LIN {X 0,Y 372.523,Z 405.276,A -85,B 0,C 180,E1 -12705.139,E2 -12705.139} C_VEL
LIN {X 0,Y 373,Z 395.69,A -85,B 0,C 180,E1 -12705.477,E2 -12705.477} C_VEL
LIN {X 0,Y 373.56,Z 352.776,A -85,B 0,C 180,E1 -12706.364,E2 -12706.364} C_VEL
LIN {X 0,Y 373.405,Z 343.149,A -85,B 0,C 180,E1 -12706.57,E2 -12706.57} C_VEL
LIN {X 0,Y 370.133,Z 321.024,A -85,B 0,C 180,E1 -12707.194,E2 -12707.194} C_VEL
LIN {X 0,Y 369.546,Z 317.373,A -85,B 0,C 180,E1 -12707.322,E2 -12707.322} C_VEL
LIN {X 0,Y 370.614,Z 302.559,A -85,B 0,C 180,E1 -12711.118,E2 -12711.118} C_VEL
LIN {X 0,Y 371.037,Z 295.89,A -85,B 0,C 180,E1 -12712.848,E2 -12712.848} C_VEL
LIN {X 0,Y 369.464,Z 286.97,A -85,B 0,C 180,E1 -12715.34,E2 -12715.34} C_VEL
LIN {X 0,Y 368.919,Z 284.344,A -85,B 0,C 180,E1 -12716.097,E2 -12716.097} C_VEL
LIN {X 0,Y 368.891,Z 284.349,A -85,B 0,C 180,E1 -12719.691,E2 -12719.691} C_VEL
LIN {X 0,Y 368.893,Z 284.348,A -85,B 0,C 180,E1 -12723.042,E2 -12723.042} C_VEL
LIN {X 0,Y 368.912,Z 284.344,A -85,B 0,C 180,E1 -12726.196,E2 -12726.196} C_VEL
LIN {X 0,Y 368.896,Z 284.351,A -85,B 0,C 180,E1 -12728.953,E2 -12728.953} C_VEL
LIN {X 0,Y 368.874,Z 284.348,A -85,B 0,C 180,E1 -12732.008,E2 -12732.008} C_VEL
LIN {X 0,Y 368.873,Z 284.351,A -85,B 0,C 180,E1 -12735.175,E2 -12735.175} C_VEL
LIN {X 0,Y 368.875,Z 284.345,A -85,B 0,C 180,E1 -12738.177,E2 -12738.177} C_VEL
LIN {X 0,Y 368.899,Z 284.348,A -85,B 0,C 180,E1 -12741.359,E2 -12741.359} C_VEL
LIN {X 0,Y 368.928,Z 284.341,A -85,B 0,C 180,E1 -12745.146,E2 -12745.146} C_VEL
LIN {X 0,Y 368.921,Z 284.338,A -85,B 0,C 180,E1 -12749.046,E2 -12749.046} C_VEL
LIN {X 0,Y 368.966,Z 284.335,A -85,B 0,C 180,E1 -12751.563,E2 -12751.563} C_VEL
LIN {X 0,Y 368.99,Z 284.33,A -85,B 0,C 180,E1 -12754.019,E2 -12754.019} C_VEL
LIN {X 0,Y 368.911,Z 284.338,A -85,B 0,C 180,E1 -12757.604,E2 -12757.604} C_VEL
LIN {X 0,Y 368.947,Z 284.337,A -85,B 0,C 180,E1 -12761.105,E2 -12761.105} C_VEL
LIN {X 0,Y 368.986,Z 284.325,A -85,B 0,C 180,E1 -12764.535,E2 -12764.535} C_VEL
LIN {X 0,Y 368.994,Z 284.332,A -85,B 0,C 180,E1 -12767.906,E2 -12767.906} C_VEL
LIN {X 0,Y 369.156,Z 284.304,A -85,B 0,C 180,E1 -12771.869,E2 -12771.869} C_VEL
LIN {X 0,Y 369.13,Z 284.317,A -85,B 0,C 180,E1 -12774.537,E2 -12774.537} C_VEL
LIN {X 0,Y 369.304,Z 284.286,A -85,B 0,C 180,E1 -12777.819,E2 -12777.819} C_VEL
LIN {X 0,Y 369.446,Z 284.273,A -85,B 0,C 180,E1 -12780,E2 -12780} C_VEL
LIN {X 0,Y 369.305,Z 284.283,A -85,B 0,C 180,E1 -12782.181,E2 -12782.181} C_VEL
LIN {X 0,Y 369.161,Z 284.309,A -85,B 0,C 180,E1 -12786.559,E2 -12786.559} C_VEL
LIN {X 0,Y 369.056,Z 284.325,A -85,B 0,C 180,E1 -12789.869,E2 -12789.869} C_VEL
LIN {X 0,Y 369.027,Z 284.331,A -85,B 0,C 180,E1 -12793.773,E2 -12793.773} C_VEL
LIN {X 0,Y 368.992,Z 284.336,A -85,B 0,C 180,E1 -12797.769,E2 -12797.769} C_VEL
LIN {X 0,Y 368.92,Z 284.341,A -85,B 0,C 180,E1 -12801.22,E2 -12801.22} C_VEL
LIN {X 0,Y 368.949,Z 284.339,A -85,B 0,C 180,E1 -12804.776,E2 -12804.776} C_VEL
LIN {X 0,Y 368.978,Z 284.334,A -85,B 0,C 180,E1 -12808.436,E2 -12808.436} C_VEL
LIN {X 0,Y 368.891,Z 284.349,A -85,B 0,C 180,E1 -12812.239,E2 -12812.239} C_VEL
LIN {X 0,Y 368.922,Z 284.338,A -85,B 0,C 180,E1 -12815.002,E2 -12815.002} C_VEL
LIN {X 0,Y 368.906,Z 284.346,A -85,B 0,C 180,E1 -12818.642,E2 -12818.642} C_VEL
LIN {X 0,Y 368.956,Z 284.341,A -85,B 0,C 180,E1 -12820.813,E2 -12820.813} C_VEL
LIN {X 0,Y 370.249,Z 291.31,A -85,B 0,C 180,E1 -12822.819,E2 -12822.819} C_VEL
LIN {X 0,Y 369.978,Z 298.523,A -85,B 0,C 180,E1 -12824.755,E2 -12824.755} C_VEL
LIN {X 0,Y 373.924,Z 318.904,A -85,B 0,C 180,E1 -12825.4,E2 -12825.4} C_VEL
LIN {X 0,Y 373.092,Z 375.949,A -85,B 0,C 180,E1 -12826.565,E2 -12826.565} C_VEL
LIN {X 0,Y 372.739,Z 386.647,A -85,B 0,C 180,E1 -12826.954,E2 -12826.954} C_VEL
LIN {X 0,Y 372.199,Z 398.56,A -85,B 0,C 180,E1 -12827.636,E2 -12827.636} C_VEL
LIN {X 0,Y 371.586,Z 407.896,A -85,B 0,C 180,E1 -12828.37,E2 -12828.37} C_VEL
LIN {X 0,Y 370.993,Z 415.935,A -85,B 0,C 180,E1 -12829.168,E2 -12829.168} C_VEL
LIN {X 0,Y 370.411,Z 422.879,A -85,B 0,C 180,E1 -12830.006,E2 -12830.006} C_VEL
LIN {X 0,Y 369.807,Z 429.621,A -85,B 0,C 180,E1 -12830.986,E2 -12830.986} C_VEL
LIN {X 0,Y 369.35,Z 434.404,A -85,B 0,C 180,E1 -12831.801,E2 -12831.801} C_VEL
LIN {X 0,Y 368.78,Z 440.973,A -85,B 0,C 180,E1 -12833.17,E2 -12833.17} C_VEL
LIN {X 0,Y 368.379,Z 445.802,A -85,B 0,C 180,E1 -12834.418,E2 -12834.418} C_VEL
LIN {X 0,Y 367.918,Z 449.947,A -85,B 0,C 180,E1 -12835.759,E2 -12835.759} C_VEL
LIN {X 0,Y 367.739,Z 453.397,A -85,B 0,C 180,E1 -12837.236,E2 -12837.236} C_VEL
LIN {X 0,Y 367.446,Z 456.117,A -85,B 0,C 180,E1 -12838.909,E2 -12838.909} C_VEL
LIN {X 0,Y 367.291,Z 457.289,A -85,B 0,C 180,E1 -12840.166,E2 -12840.166} C_VEL
LIN {X 0,Y 367.214,Z 457.874,A -85,B 0,C 180,E1 -12841.689,E2 -12841.689} C_VEL
LIN {X 0,Y 367.2,Z 457.67,A -85,B 0,C 180,E1 -12842.656,E2 -12842.656} C_VEL
LIN {X 0,Y 367.282,Z 456.753,A -85,B 0,C 180,E1 -12844.074,E2 -12844.074} C_VEL
LIN {X 0,Y 367.469,Z 454.638,A -85,B 0,C 180,E1 -12845.721,E2 -12845.721} C_VEL
LIN {X 0,Y 367.777,Z 450.863,A -85,B 0,C 180,E1 -12847.532,E2 -12847.532} C_VEL
LIN {X 0,Y 368.018,Z 447.468,A -85,B 0,C 180,E1 -12848.726,E2 -12848.726} C_VEL
LIN {X 0,Y 368.416,Z 442.007,A -85,B 0,C 180,E1 -12850.209,E2 -12850.209} C_VEL
LIN {X 0,Y 368.818,Z 436.622,A -85,B 0,C 180,E1 -12851.388,E2 -12851.388} C_VEL
LIN {X 0,Y 369.347,Z 430.05,A -85,B 0,C 180,E1 -12852.561,E2 -12852.561} C_VEL
LIN {X 0,Y 369.885,Z 423.088,A -85,B 0,C 180,E1 -12853.583,E2 -12853.583} C_VEL
LIN {X 0,Y 370.406,Z 415.905,A -85,B 0,C 180,E1 -12854.455,E2 -12854.455} C_VEL
LIN {X 0,Y 370.966,Z 408.076,A -85,B 0,C 180,E1 -12855.234,E2 -12855.234} C_VEL
LIN {X 0,Y 371.424,Z 399.77,A -85,B 0,C 180,E1 -12855.9,E2 -12855.9} C_VEL
LIN {X 0,Y 371.823,Z 390.588,A -85,B 0,C 180,E1 -12856.473,E2 -12856.473} C_VEL
LIN {X 0,Y 372.259,Z 379.24,A -85,B 0,C 180,E1 -12856.976,E2 -12856.976} C_VEL
LIN {X 0,Y 372.545,Z 362.521,A -85,B 0,C 180,E1 -12857.367,E2 -12857.367} C_VEL
LIN {X 0,Y 372.968,Z 318.576,A -85,B 0,C 180,E1 -12858.237,E2 -12858.237} C_VEL
LIN {X 0,Y 369.543,Z 298.791,A -85,B 0,C 180,E1 -12858.8,E2 -12858.8} C_VEL
LIN {X 0,Y 369.932,Z 290.475,A -85,B 0,C 180,E1 -12861.258,E2 -12861.258} C_VEL
LIN {X 0,Y 369.217,Z 284.308,A -85,B 0,C 180,E1 -12863.168,E2 -12863.168} C_VEL
LIN {X 0,Y 369.318,Z 284.296,A -85,B 0,C 180,E1 -12867.819,E2 -12867.819} C_VEL
LIN {X 0,Y 369.459,Z 284.278,A -85,B 0,C 180,E1 -12870,E2 -12870} C_VEL
LIN {X 0,Y 369.319,Z 284.294,A -85,B 0,C 180,E1 -12872.181,E2 -12872.181} C_VEL
LIN {X 0,Y 369.18,Z 284.309,A -85,B 0,C 180,E1 -12876.558,E2 -12876.558} C_VEL
LIN {X 0,Y 369.068,Z 284.323,A -85,B 0,C 180,E1 -12879.868,E2 -12879.868} C_VEL
LIN {X 0,Y 369.038,Z 284.325,A -85,B 0,C 180,E1 -12883.772,E2 -12883.772} C_VEL
LIN {X 0,Y 369.01,Z 284.333,A -85,B 0,C 180,E1 -12884.425,E2 -12884.425} C_VEL
LIN {X 0,Y 368.294,Z 284.417,A -85,B 0,C 180,E1 -12885.335,E2 -12885.335} C_VEL
LIN {X 0,Y 365.388,Z 284.782,A -85,B 0,C 180,E1 -12886.815,E2 -12886.815} C_VEL
LIN {X 0,Y 362.968,Z 285.082,A -85,B 0,C 180,E1 -12888.013,E2 -12888.013} C_VEL
LIN {X 0,Y 361.955,Z 285.21,A -85,B 0,C 180,E1 -12888.939,E2 -12888.939} C_VEL
LIN {X 0,Y 361.885,Z 285.216,A -85,B 0,C 180,E1 -12889.253,E2 -12889.253} C_VEL
LIN {X 0,Y 361.882,Z 285.221,A -85,B 0,C 180,E1 -12892.855,E2 -12892.855} C_VEL
LIN {X 0,Y 361.94,Z 285.214,A -85,B 0,C 180,E1 -12896.721,E2 -12896.721} C_VEL
LIN {X 0,Y 361.873,Z 285.218,A -85,B 0,C 180,E1 -12900.327,E2 -12900.327} C_VEL
LIN {X 0,Y 361.851,Z 285.22,A -85,B 0,C 180,E1 -12904.28,E2 -12904.28} C_VEL
LIN {X 0,Y 361.86,Z 285.226,A -85,B 0,C 180,E1 -12907.222,E2 -12907.222} C_VEL
LIN {X 0,Y 361.832,Z 285.223,A -85,B 0,C 180,E1 -12910.754,E2 -12910.754} C_VEL
LIN {X 0,Y 361.841,Z 285.221,A -85,B 0,C 180,E1 -12914.363,E2 -12914.363} C_VEL
LIN {X 0,Y 361.884,Z 285.222,A -85,B 0,C 180,E1 -12917.558,E2 -12917.558} C_VEL
LIN {X 0,Y 361.868,Z 285.218,A -85,B 0,C 180,E1 -12920.972,E2 -12920.972} C_VEL
LIN {X 0,Y 361.868,Z 285.218,A -85,B 0,C 180,E1 -12924.654,E2 -12924.654} C_VEL
LIN {X 0,Y 361.831,Z 285.225,A -85,B 0,C 180,E1 -12928.37,E2 -12928.37} C_VEL
LIN {X 0,Y 361.894,Z 285.214,A -85,B 0,C 180,E1 -12930.955,E2 -12930.955} C_VEL
LIN {X 0,Y 361.946,Z 285.208,A -85,B 0,C 180,E1 -12933.474,E2 -12933.474} C_VEL
LIN {X 0,Y 361.881,Z 285.216,A -85,B 0,C 180,E1 -12937.144,E2 -12937.144} C_VEL
LIN {X 0,Y 361.895,Z 285.218,A -85,B 0,C 180,E1 -12940.723,E2 -12940.723} C_VEL
LIN {X 0,Y 361.923,Z 285.212,A -85,B 0,C 180,E1 -12943.065,E2 -12943.065} C_VEL
LIN {X 0,Y 361.989,Z 285.208,A -85,B 0,C 180,E1 -12946.527,E2 -12946.527} C_VEL
LIN {X 0,Y 362.021,Z 285.199,A -85,B 0,C 180,E1 -12949.938,E2 -12949.938} C_VEL
LIN {X 0,Y 362.151,Z 285.184,A -85,B 0,C 180,E1 -12953.313,E2 -12953.313} C_VEL
LIN {X 0,Y 362.271,Z 285.168,A -85,B 0,C 180,E1 -12957.776,E2 -12957.776} C_VEL
LIN {X 0,Y 362.416,Z 285.149,A -85,B 0,C 180,E1 -12960,E2 -12960} C_VEL
LIN {X 0,Y 362.269,Z 285.167,A -85,B 0,C 180,E1 -12962.223,E2 -12962.223} C_VEL
LIN {X 0,Y 362.151,Z 285.183,A -85,B 0,C 180,E1 -12966.686,E2 -12966.686} C_VEL
LIN {X 0,Y 362.024,Z 285.199,A -85,B 0,C 180,E1 -12970.062,E2 -12970.062} C_VEL
LIN {X 0,Y 361.988,Z 285.206,A -85,B 0,C 180,E1 -12973.899,E2 -12973.899} C_VEL
LIN {X 0,Y 361.958,Z 285.211,A -85,B 0,C 180,E1 -12977.939,E2 -12977.939} C_VEL
LIN {X 0,Y 361.871,Z 285.221,A -85,B 0,C 180,E1 -12981.654,E2 -12981.654} C_VEL
LIN {X 0,Y 361.917,Z 285.212,A -85,B 0,C 180,E1 -12985.291,E2 -12985.291} C_VEL
LIN {X 0,Y 361.899,Z 285.217,A -85,B 0,C 180,E1 -12987.78,E2 -12987.78} C_VEL
LIN {X 0,Y 361.829,Z 285.223,A -85,B 0,C 180,E1 -12991.63,E2 -12991.63} C_VEL
LIN {X 0,Y 361.866,Z 285.218,A -85,B 0,C 180,E1 -12995.345,E2 -12995.345} C_VEL
LIN {X 0,Y 361.86,Z 285.22,A -85,B 0,C 180,E1 -12999.027,E2 -12999.027} C_VEL
LIN {X 0,Y 361.829,Z 285.227,A -85,B 0,C 180,E1 -13002.83,E2 -13002.83} C_VEL
LIN {X 0,Y 361.813,Z 285.225,A -85,B 0,C 180,E1 -13005.947,E2 -13005.947} C_VEL
LIN {X 0,Y 361.829,Z 285.225,A -85,B 0,C 180,E1 -13009.246,E2 -13009.246} C_VEL
LIN {X 0,Y 361.858,Z 285.223,A -85,B 0,C 180,E1 -13012.778,E2 -13012.778} C_VEL
LIN {X 0,Y 361.85,Z 285.221,A -85,B 0,C 180,E1 -13015.72,E2 -13015.72} C_VEL
LIN {X 0,Y 361.861,Z 285.22,A -85,B 0,C 180,E1 -13019.672,E2 -13019.672} C_VEL
LIN {X 0,Y 361.874,Z 285.222,A -85,B 0,C 180,E1 -13023.78,E2 -13023.78} C_VEL
LIN {X 0,Y 361.907,Z 285.404,A -85,B 0,C 180,E1 -13023.938,E2 -13023.938} C_VEL
LIN {X 0,Y 363.844,Z 295.855,A -85,B 0,C 180,E1 -13026.975,E2 -13026.975} C_VEL
LIN {X 0,Y 363.495,Z 302.362,A -85,B 0,C 180,E1 -13028.746,E2 -13028.746} C_VEL
LIN {X 0,Y 362.389,Z 316.398,A -85,B 0,C 180,E1 -13032.507,E2 -13032.507} C_VEL
LIN {X 0,Y 362.291,Z 317.88,A -85,B 0,C 180,E1 -13032.902,E2 -13032.902} C_VEL
LIN {X 0,Y 366.001,Z 345.967,A -85,B 0,C 180,E1 -13033.672,E2 -13033.672} C_VEL
LIN {X 0,Y 365.308,Z 395.497,A -85,B 0,C 180,E1 -13034.697,E2 -13034.697} C_VEL
LIN {X 0,Y 364.866,Z 405.848,A -85,B 0,C 180,E1 -13035.071,E2 -13035.071} C_VEL
LIN {X 0,Y 364.198,Z 417.985,A -85,B 0,C 180,E1 -13035.757,E2 -13035.757} C_VEL
LIN {X 0,Y 363.671,Z 426.806,A -85,B 0,C 180,E1 -13036.449,E2 -13036.449} C_VEL
LIN {X 0,Y 363.046,Z 435.21,A -85,B 0,C 180,E1 -13037.279,E2 -13037.279} C_VEL
LIN {X 0,Y 362.479,Z 443.159,A -85,B 0,C 180,E1 -13038.254,E2 -13038.254} C_VEL
LIN {X 0,Y 361.867,Z 450.582,A -85,B 0,C 180,E1 -13039.368,E2 -13039.368} C_VEL
LIN {X 0,Y 361.242,Z 458.107,A -85,B 0,C 180,E1 -13040.764,E2 -13040.764} C_VEL
LIN {X 0,Y 360.844,Z 464.009,A -85,B 0,C 180,E1 -13042.164,E2 -13042.164} C_VEL
LIN {X 0,Y 360.609,Z 467.845,A -85,B 0,C 180,E1 -13043.285,E2 -13043.285} C_VEL
LIN {X 0,Y 360.429,Z 472.249,A -85,B 0,C 180,E1 -13044.966,E2 -13044.966} C_VEL
LIN {X 0,Y 360.318,Z 475.324,A -85,B 0,C 180,E1 -13046.646,E2 -13046.646} C_VEL
LIN {X 0,Y 360.269,Z 476.725,A -85,B 0,C 180,E1 -13047.764,E2 -13047.764} C_VEL
LIN {X 0,Y 360.302,Z 477.636,A -85,B 0,C 180,E1 -13048.882,E2 -13048.882} C_VEL
LIN {X 0,Y 360.357,Z 477.957,A -85,B 0,C 180,E1 -13050,E2 -13050} C_VEL
LIN {X 0,Y 360.301,Z 477.756,A -85,B 0,C 180,E1 -13051.118,E2 -13051.118} C_VEL
LIN {X 0,Y 360.267,Z 477.089,A -85,B 0,C 180,E1 -13052.236,E2 -13052.236} C_VEL
LIN {X 0,Y 360.317,Z 475.947,A -85,B 0,C 180,E1 -13053.354,E2 -13053.354} C_VEL
LIN {X 0,Y 360.424,Z 474.277,A -85,B 0,C 180,E1 -13054.473,E2 -13054.473} C_VEL
LIN {X 0,Y 360.51,Z 470.594,A -85,B 0,C 180,E1 -13056.162,E2 -13056.162} C_VEL
LIN {X 0,Y 360.801,Z 467.472,A -85,B 0,C 180,E1 -13057.274,E2 -13057.274} C_VEL
LIN {X 0,Y 361.128,Z 462.472,A -85,B 0,C 180,E1 -13058.674,E2 -13058.674} C_VEL
LIN {X 0,Y 361.678,Z 456.185,A -85,B 0,C 180,E1 -13060.072,E2 -13060.072} C_VEL
LIN {X 0,Y 362.293,Z 450.045,A -85,B 0,C 180,E1 -13061.185,E2 -13061.185} C_VEL
LIN {X 0,Y 362.863,Z 443.608,A -85,B 0,C 180,E1 -13062.159,E2 -13062.159} C_VEL
LIN {X 0,Y 363.565,Z 435.824,A -85,B 0,C 180,E1 -13063.128,E2 -13063.128} C_VEL
LIN {X 0,Y 364.254,Z 427.639,A -85,B 0,C 180,E1 -13063.956,E2 -13063.956} C_VEL
LIN {X 0,Y 365.019,Z 417.265,A -85,B 0,C 180,E1 -13064.78,E2 -13064.78} C_VEL
LIN {X 0,Y 365.679,Z 405.709,A -85,B 0,C 180,E1 -13065.43,E2 -13065.43} C_VEL
LIN {X 0,Y 366.207,Z 395.084,A -85,B 0,C 180,E1 -13065.811,E2 -13065.811} C_VEL
LIN {X 0,Y 366.788,Z 344.866,A -85,B 0,C 180,E1 -13066.868,E2 -13066.868} C_VEL
LIN {X 0,Y 363.324,Z 321.428,A -85,B 0,C 180,E1 -13067.552,E2 -13067.552} C_VEL
LIN {X 0,Y 362.599,Z 317.17,A -85,B 0,C 180,E1 -13067.701,E2 -13067.701} C_VEL
LIN {X 0,Y 363.744,Z 302.471,A -85,B 0,C 180,E1 -13071.536,E2 -13071.536} C_VEL
LIN {X 0,Y 364.042,Z 296.917,A -85,B 0,C 180,E1 -13073.012,E2 -13073.012} C_VEL
LIN {X 0,Y 362.423,Z 288.013,A -85,B 0,C 180,E1 -13075.56,E2 -13075.56} C_VEL
LIN {X 0,Y 361.86,Z 285.224,A -85,B 0,C 180,E1 -13076.376,E2 -13076.376} C_VEL
LIN {X 0,Y 361.852,Z 285.228,A -85,B 0,C 180,E1 -13080.329,E2 -13080.329} C_VEL
LIN {X 0,Y 361.85,Z 285.223,A -85,B 0,C 180,E1 -13084.28,E2 -13084.28} C_VEL
LIN {X 0,Y 361.858,Z 285.226,A -85,B 0,C 180,E1 -13087.222,E2 -13087.222} C_VEL
LIN {X 0,Y 361.829,Z 285.232,A -85,B 0,C 180,E1 -13090.754,E2 -13090.754} C_VEL
LIN {X 0,Y 361.81,Z 285.23,A -85,B 0,C 180,E1 -13094.368,E2 -13094.368} C_VEL
LIN {X 0,Y 361.829,Z 285.227,A -85,B 0,C 180,E1 -13097.567,E2 -13097.567} C_VEL
LIN {X 0,Y 361.86,Z 285.222,A -85,B 0,C 180,E1 -13100.973,E2 -13100.973} C_VEL
LIN {X 0,Y 361.866,Z 285.219,A -85,B 0,C 180,E1 -13104.655,E2 -13104.655} C_VEL
LIN {X 0,Y 361.829,Z 285.223,A -85,B 0,C 180,E1 -13108.37,E2 -13108.37} C_VEL
LIN {X 0,Y 361.892,Z 285.214,A -85,B 0,C 180,E1 -13110.955,E2 -13110.955} C_VEL
LIN {X 0,Y 361.944,Z 285.202,A -85,B 0,C 180,E1 -13113.474,E2 -13113.474} C_VEL
LIN {X 0,Y 361.869,Z 285.214,A -85,B 0,C 180,E1 -13117.143,E2 -13117.143} C_VEL
LIN {X 0,Y 361.894,Z 285.217,A -85,B 0,C 180,E1 -13120.723,E2 -13120.723} C_VEL
LIN {X 0,Y 361.922,Z 285.207,A -85,B 0,C 180,E1 -13123.066,E2 -13123.066} C_VEL
LIN {X 0,Y 361.988,Z 285.206,A -85,B 0,C 180,E1 -13126.528,E2 -13126.528} C_VEL
LIN {X 0,Y 362.02,Z 285.195,A -85,B 0,C 180,E1 -13129.938,E2 -13129.938} C_VEL
LIN {X 0,Y 362.152,Z 285.183,A -85,B 0,C 180,E1 -13133.314,E2 -13133.314} C_VEL
LIN {X 0,Y 362.268,Z 285.163,A -85,B 0,C 180,E1 -13137.776,E2 -13137.776} C_VEL
LIN {X 0,Y 362.416,Z 285.149,A -85,B 0,C 180,E1 -13140,E2 -13140} C_VEL
LIN {X 0,Y 362.269,Z 285.159,A -85,B 0,C 180,E1 -13142.224,E2 -13142.224} C_VEL
LIN {X 0,Y 362.123,Z 285.187,A -85,B 0,C 180,E1 -13146.687,E2 -13146.687} C_VEL
LIN {X 0,Y 362.02,Z 285.201,A -85,B 0,C 180,E1 -13150.062,E2 -13150.062} C_VEL
LIN {X 0,Y 361.988,Z 285.207,A -85,B 0,C 180,E1 -13153.899,E2 -13153.899} C_VEL
LIN {X 0,Y 361.958,Z 285.213,A -85,B 0,C 180,E1 -13157.939,E2 -13157.939} C_VEL
LIN {X 0,Y 361.883,Z 285.222,A -85,B 0,C 180,E1 -13161.654,E2 -13161.654} C_VEL
LIN {X 0,Y 361.919,Z 285.216,A -85,B 0,C 180,E1 -13165.291,E2 -13165.291} C_VEL
LIN {X 0,Y 361.914,Z 285.218,A -85,B 0,C 180,E1 -13167.779,E2 -13167.779} C_VEL
LIN {X 0,Y 361.839,Z 285.223,A -85,B 0,C 180,E1 -13171.286,E2 -13171.286} C_VEL
LIN {X 0,Y 361.847,Z 285.223,A -85,B 0,C 180,E1 -13174.281,E2 -13174.281} C_VEL
LIN {X 0,Y 361.859,Z 285.223,A -85,B 0,C 180,E1 -13177.224,E2 -13177.224} C_VEL
LIN {X 0,Y 361.958,Z 285.413,A -85,B 0,C 180,E1 -13180.592,E2 -13180.592} C_VEL
LIN {X 0,Y 363.312,Z 292.544,A -85,B 0,C 180,E1 -13182.688,E2 -13182.688} C_VEL
LIN {X 0,Y 363.067,Z 298.691,A -85,B 0,C 180,E1 -13184.372,E2 -13184.372} C_VEL
LIN {X 0,Y 367.17,Z 319.733,A -85,B 0,C 180,E1 -13185.064,E2 -13185.064} C_VEL
LIN {X 0,Y 366.309,Z 376.155,A -85,B 0,C 180,E1 -13186.241,E2 -13186.241} C_VEL
LIN {X 0,Y 365.954,Z 386.701,A -85,B 0,C 180,E1 -13186.632,E2 -13186.632} C_VEL
LIN {X 0,Y 365.456,Z 397.63,A -85,B 0,C 180,E1 -13187.25,E2 -13187.25} C_VEL
LIN {X 0,Y 364.87,Z 406.864,A -85,B 0,C 180,E1 -13187.969,E2 -13187.969} C_VEL
LIN {X 0,Y 364.187,Z 415.457,A -85,B 0,C 180,E1 -13188.817,E2 -13188.817} C_VEL
LIN {X 0,Y 363.563,Z 422.314,A -85,B 0,C 180,E1 -13189.642,E2 -13189.642} C_VEL
LIN {X 0,Y 362.919,Z 428.888,A -85,B 0,C 180,E1 -13190.59,E2 -13190.59} C_VEL
LIN {X 0,Y 362.355,Z 434.922,A -85,B 0,C 180,E1 -13191.638,E2 -13191.638} C_VEL
LIN {X 0,Y 361.791,Z 441.194,A -85,B 0,C 180,E1 -13192.974,E2 -13192.974} C_VEL
LIN {X 0,Y 361.4,Z 445.075,A -85,B 0,C 180,E1 -13193.968,E2 -13193.968} C_VEL
LIN {X 0,Y 361.027,Z 449.08,A -85,B 0,C 180,E1 -13195.215,E2 -13195.215} C_VEL
LIN {X 0,Y 360.766,Z 451.885,A -85,B 0,C 180,E1 -13196.277,E2 -13196.277} C_VEL
LIN {X 0,Y 360.607,Z 454.538,A -85,B 0,C 180,E1 -13197.592,E2 -13197.592} C_VEL
LIN {X 0,Y 360.282,Z 456.997,A -85,B 0,C 180,E1 -13199.525,E2 -13199.525} C_VEL
LIN {X 0,Y 360.117,Z 458.011,A -85,B 0,C 180,E1 -13201.428,E2 -13201.428} C_VEL
LIN {X 0,Y 360.137,Z 457.601,A -85,B 0,C 180,E1 -13203.332,E2 -13203.332} C_VEL
LIN {X 0,Y 360.222,Z 456.505,A -85,B 0,C 180,E1 -13204.583,E2 -13204.583} C_VEL
LIN {X 0,Y 360.514,Z 453.728,A -85,B 0,C 180,E1 -13206.382,E2 -13206.382} C_VEL
LIN {X 0,Y 360.718,Z 450.886,A -85,B 0,C 180,E1 -13207.672,E2 -13207.672} C_VEL
LIN {X 0,Y 361.028,Z 446.618,A -85,B 0,C 180,E1 -13209.132,E2 -13209.132} C_VEL
LIN {X 0,Y 361.382,Z 441.942,A -85,B 0,C 180,E1 -13210.4,E2 -13210.4} C_VEL
LIN {X 0,Y 361.832,Z 436.493,A -85,B 0,C 180,E1 -13211.602,E2 -13211.602} C_VEL
LIN {X 0,Y 362.37,Z 429.854,A -85,B 0,C 180,E1 -13212.799,E2 -13212.799} C_VEL
LIN {X 0,Y 362.917,Z 422.836,A -85,B 0,C 180,E1 -13213.837,E2 -13213.837} C_VEL
LIN {X 0,Y 363.499,Z 415.501,A -85,B 0,C 180,E1 -13214.731,E2 -13214.731} C_VEL
LIN {X 0,Y 364.145,Z 406.579,A -85,B 0,C 180,E1 -13215.612,E2 -13215.612} C_VEL
LIN {X 0,Y 364.748,Z 394.797,A -85,B 0,C 180,E1 -13216.49,E2 -13216.49} C_VEL
LIN {X 0,Y 365.134,Z 385.095,A -85,B 0,C 180,E1 -13217,E2 -13217} C_VEL
LIN {X 0,Y 365.418,Z 376.079,A -85,B 0,C 180,E1 -13217.328,E2 -13217.328} C_VEL
LIN {X 0,Y 365.997,Z 335.574,A -85,B 0,C 180,E1 -13218.175,E2 -13218.175} C_VEL
LIN {X 0,Y 366.158,Z 319.703,A -85,B 0,C 180,E1 -13218.496,E2 -13218.496} C_VEL
LIN {X 0,Y 362.555,Z 298.937,A -85,B 0,C 180,E1 -13219.106,E2 -13219.106} C_VEL
LIN {X 0,Y 362.939,Z 292.344,A -85,B 0,C 180,E1 -13221.089,E2 -13221.089} C_VEL
LIN {X 0,Y 362.186,Z 285.185,A -85,B 0,C 180,E1 -13223.349,E2 -13223.349} C_VEL
LIN {X 0,Y 362.282,Z 285.172,A -85,B 0,C 180,E1 -13227.777,E2 -13227.777} C_VEL
LIN {X 0,Y 362.428,Z 285.154,A -85,B 0,C 180,E1 -13230,E2 -13230} C_VEL
LIN {X 0,Y 362.283,Z 285.17,A -85,B 0,C 180,E1 -13232.223,E2 -13232.223} C_VEL
LIN {X 0,Y 362.141,Z 285.185,A -85,B 0,C 180,E1 -13236.687,E2 -13236.687} C_VEL
LIN {X 0,Y 362.032,Z 285.202,A -85,B 0,C 180,E1 -13240.062,E2 -13240.062} C_VEL
LIN {X 0,Y 361.999,Z 285.203,A -85,B 0,C 180,E1 -13243.898,E2 -13243.898} C_VEL
LIN {X 0,Y 361.929,Z 285.212,A -85,B 0,C 180,E1 -13246.934,E2 -13246.934} C_VEL
LIN {X 0,Y 361.885,Z 285.216,A -85,B 0,C 180,E1 -13249.253,E2 -13249.253} C_VEL
LIN {X 0,Y 361.239,Z 285.301,A -85,B 0,C 180,E1 -13250.182,E2 -13250.182} C_VEL
LIN {X 0,Y 358.356,Z 285.657,A -85,B 0,C 180,E1 -13251.691,E2 -13251.691} C_VEL
LIN {X 0,Y 355.921,Z 285.963,A -85,B 0,C 180,E1 -13252.912,E2 -13252.912} C_VEL
LIN {X 0,Y 354.909,Z 286.085,A -85,B 0,C 180,E1 -13253.858,E2 -13253.858} C_VEL
LIN {X 0,Y 354.845,Z 286.093,A -85,B 0,C 180,E1 -13254.178,E2 -13254.178} C_VEL
LIN {X 0,Y 354.882,Z 286.092,A -85,B 0,C 180,E1 -13257.095,E2 -13257.095} C_VEL
LIN {X 0,Y 354.852,Z 286.092,A -85,B 0,C 180,E1 -13259.678,E2 -13259.678} C_VEL
LIN {X 0,Y 354.804,Z 286.099,A -85,B 0,C 180,E1 -13263.701,E2 -13263.701} C_VEL
LIN {X 0,Y 354.794,Z 286.099,A -85,B 0,C 180,E1 -13266.459,E2 -13266.459} C_VEL
LIN {X 0,Y 354.821,Z 286.101,A -85,B 0,C 180,E1 -13269.423,E2 -13269.423} C_VEL
LIN {X 0,Y 354.786,Z 286.101,A -85,B 0,C 180,E1 -13272.867,E2 -13272.867} C_VEL
LIN {X 0,Y 354.835,Z 286.095,A -85,B 0,C 180,E1 -13276.114,E2 -13276.114} C_VEL
LIN {X 0,Y 354.852,Z 286.093,A -85,B 0,C 180,E1 -13279.188,E2 -13279.188} C_VEL
LIN {X 0,Y 354.803,Z 286.099,A -85,B 0,C 180,E1 -13282.401,E2 -13282.401} C_VEL
LIN {X 0,Y 354.805,Z 286.097,A -85,B 0,C 180,E1 -13284.94,E2 -13284.94} C_VEL
LIN {X 0,Y 354.786,Z 286.102,A -85,B 0,C 180,E1 -13288.404,E2 -13288.404} C_VEL
LIN {X 0,Y 354.846,Z 286.094,A -85,B 0,C 180,E1 -13291.618,E2 -13291.618} C_VEL
LIN {X 0,Y 354.891,Z 286.094,A -85,B 0,C 180,E1 -13294.172,E2 -13294.172} C_VEL
LIN {X 0,Y 354.826,Z 286.097,A -85,B 0,C 180,E1 -13297.893,E2 -13297.893} C_VEL
LIN {X 0,Y 354.913,Z 286.085,A -85,B 0,C 180,E1 -13301.891,E2 -13301.891} C_VEL
LIN {X 0,Y 354.933,Z 286.082,A -85,B 0,C 180,E1 -13305.981,E2 -13305.981} C_VEL
LIN {X 0,Y 354.967,Z 286.077,A -85,B 0,C 180,E1 -13309.735,E2 -13309.735} C_VEL
LIN {X 0,Y 355.115,Z 286.062,A -85,B 0,C 180,E1 -13313.18,E2 -13313.18} C_VEL
LIN {X 0,Y 355.234,Z 286.044,A -85,B 0,C 180,E1 -13317.732,E2 -13317.732} C_VEL
LIN {X 0,Y 355.386,Z 286.025,A -85,B 0,C 180,E1 -13320,E2 -13320} C_VEL
LIN {X 0,Y 355.232,Z 286.044,A -85,B 0,C 180,E1 -13322.268,E2 -13322.268} C_VEL
LIN {X 0,Y 355.114,Z 286.06,A -85,B 0,C 180,E1 -13326.82,E2 -13326.82} C_VEL
LIN {X 0,Y 354.971,Z 286.077,A -85,B 0,C 180,E1 -13330.264,E2 -13330.264} C_VEL
LIN {X 0,Y 354.933,Z 286.084,A -85,B 0,C 180,E1 -13334.019,E2 -13334.019} C_VEL
LIN {X 0,Y 354.913,Z 286.087,A -85,B 0,C 180,E1 -13338.109,E2 -13338.109} C_VEL
LIN {X 0,Y 354.817,Z 286.1,A -85,B 0,C 180,E1 -13342.107,E2 -13342.107} C_VEL
LIN {X 0,Y 354.889,Z 286.091,A -85,B 0,C 180,E1 -13345.828,E2 -13345.828} C_VEL
LIN {X 0,Y 354.809,Z 286.099,A -85,B 0,C 180,E1 -13349.683,E2 -13349.683} C_VEL
LIN {X 0,Y 354.798,Z 286.099,A -85,B 0,C 180,E1 -13353.703,E2 -13353.703} C_VEL
LIN {X 0,Y 354.79,Z 286.105,A -85,B 0,C 180,E1 -13356.46,E2 -13356.46} C_VEL
LIN {X 0,Y 354.817,Z 286.096,A -85,B 0,C 180,E1 -13359.424,E2 -13359.424} C_VEL
LIN {X 0,Y 354.781,Z 286.104,A -85,B 0,C 180,E1 -13362.868,E2 -13362.868} C_VEL
LIN {X 0,Y 354.762,Z 286.104,A -85,B 0,C 180,E1 -13366.104,E2 -13366.104} C_VEL
LIN {X 0,Y 354.781,Z 286.103,A -85,B 0,C 180,E1 -13369.18,E2 -13369.18} C_VEL
LIN {X 0,Y 354.802,Z 286.099,A -85,B 0,C 180,E1 -13372.404,E2 -13372.404} C_VEL
LIN {X 0,Y 354.808,Z 286.103,A -85,B 0,C 180,E1 -13374.942,E2 -13374.942} C_VEL
LIN {X 0,Y 354.789,Z 286.1,A -85,B 0,C 180,E1 -13378.406,E2 -13378.406} C_VEL
LIN {X 0,Y 354.798,Z 286.103,A -85,B 0,C 180,E1 -13381.615,E2 -13381.615} C_VEL
LIN {X 0,Y 354.852,Z 286.176,A -85,B 0,C 180,E1 -13383.696,E2 -13383.696} C_VEL
LIN {X 0,Y 356.803,Z 296.623,A -85,B 0,C 180,E1 -13386.801,E2 -13386.801} C_VEL
LIN {X 0,Y 356.623,Z 302.05,A -85,B 0,C 180,E1 -13388.315,E2 -13388.315} C_VEL
LIN {X 0,Y 355.423,Z 316.087,A -85,B 0,C 180,E1 -13392.153,E2 -13392.153} C_VEL
LIN {X 0,Y 355.295,Z 317.805,A -85,B 0,C 180,E1 -13392.62,E2 -13392.62} C_VEL
LIN {X 0,Y 359.124,Z 346.713,A -85,B 0,C 180,E1 -13393.403,E2 -13393.403} C_VEL
LIN {X 0,Y 358.424,Z 395.401,A -85,B 0,C 180,E1 -13394.432,E2 -13394.432} C_VEL
LIN {X 0,Y 357.939,Z 405.711,A -85,B 0,C 180,E1 -13394.812,E2 -13394.812} C_VEL
LIN {X 0,Y 357.306,Z 417.356,A -85,B 0,C 180,E1 -13395.476,E2 -13395.476} C_VEL
LIN {X 0,Y 356.765,Z 426.263,A -85,B 0,C 180,E1 -13396.182,E2 -13396.182} C_VEL
LIN {X 0,Y 356.09,Z 434.729,A -85,B 0,C 180,E1 -13397.027,E2 -13397.027} C_VEL
LIN {X 0,Y 355.485,Z 442.726,A -85,B 0,C 180,E1 -13398.019,E2 -13398.019} C_VEL
LIN {X 0,Y 354.863,Z 450.19,A -85,B 0,C 180,E1 -13399.156,E2 -13399.156} C_VEL
LIN {X 0,Y 354.224,Z 457.753,A -85,B 0,C 180,E1 -13400.579,E2 -13400.579} C_VEL
LIN {X 0,Y 353.786,Z 463.701,A -85,B 0,C 180,E1 -13402.007,E2 -13402.007} C_VEL
LIN {X 0,Y 353.537,Z 467.549,A -85,B 0,C 180,E1 -13403.15,E2 -13403.15} C_VEL
LIN {X 0,Y 353.329,Z 471.989,A -85,B 0,C 180,E1 -13404.865,E2 -13404.865} C_VEL
LIN {X 0,Y 353.241,Z 475.083,A -85,B 0,C 180,E1 -13406.578,E2 -13406.578} C_VEL
LIN {X 0,Y 353.177,Z 476.503,A -85,B 0,C 180,E1 -13407.719,E2 -13407.719} C_VEL
LIN {X 0,Y 353.202,Z 477.424,A -85,B 0,C 180,E1 -13408.86,E2 -13408.86} C_VEL
LIN {X 0,Y 353.26,Z 477.751,A -85,B 0,C 180,E1 -13410,E2 -13410} C_VEL
LIN {X 0,Y 353.201,Z 477.567,A -85,B 0,C 180,E1 -13411.14,E2 -13411.14} C_VEL
LIN {X 0,Y 353.175,Z 476.916,A -85,B 0,C 180,E1 -13412.281,E2 -13412.281} C_VEL
LIN {X 0,Y 353.241,Z 475.791,A -85,B 0,C 180,E1 -13413.422,E2 -13413.422} C_VEL
LIN {X 0,Y 353.341,Z 473.002,A -85,B 0,C 180,E1 -13415.135,E2 -13415.135} C_VEL
LIN {X 0,Y 353.404,Z 470.949,A -85,B 0,C 180,E1 -13416.106,E2 -13416.106} C_VEL
LIN {X 0,Y 353.734,Z 467.362,A -85,B 0,C 180,E1 -13417.42,E2 -13417.42} C_VEL
LIN {X 0,Y 354.095,Z 462.388,A -85,B 0,C 180,E1 -13418.848,E2 -13418.848} C_VEL
LIN {X 0,Y 354.679,Z 456.124,A -85,B 0,C 180,E1 -13420.272,E2 -13420.272} C_VEL
LIN {X 0,Y 355.321,Z 450.018,A -85,B 0,C 180,E1 -13421.408,E2 -13421.408} C_VEL
LIN {X 0,Y 355.924,Z 443.624,A -85,B 0,C 180,E1 -13422.4,E2 -13422.4} C_VEL
LIN {X 0,Y 356.67,Z 435.893,A -85,B 0,C 180,E1 -13423.387,E2 -13423.387} C_VEL
LIN {X 0,Y 357.387,Z 427.777,A -85,B 0,C 180,E1 -13424.229,E2 -13424.229} C_VEL
LIN {X 0,Y 358.031,Z 419.367,A -85,B 0,C 180,E1 -13424.929,E2 -13424.929} C_VEL
LIN {X 0,Y 358.685,Z 409.576,A -85,B 0,C 180,E1 -13425.556,E2 -13425.556} C_VEL
LIN {X 0,Y 359.368,Z 397.423,A -85,B 0,C 180,E1 -13426.083,E2 -13426.083} C_VEL
LIN {X 0,Y 359.804,Z 376.745,A -85,B 0,C 180,E1 -13426.557,E2 -13426.557} C_VEL
LIN {X 0,Y 359.972,Z 344.736,A -85,B 0,C 180,E1 -13427.234,E2 -13427.234} C_VEL
LIN {X 0,Y 356.153,Z 319.819,A -85,B 0,C 180,E1 -13427.989,E2 -13427.989} C_VEL
LIN {X 0,Y 355.668,Z 316.958,A -85,B 0,C 180,E1 -13428.095,E2 -13428.095} C_VEL
LIN {X 0,Y 356.885,Z 302.417,A -85,B 0,C 180,E1 -13431.972,E2 -13431.972} C_VEL
LIN {X 0,Y 357.053,Z 297.977,A -85,B 0,C 180,E1 -13433.182,E2 -13433.182} C_VEL
LIN {X 0,Y 355.409,Z 289.071,A -85,B 0,C 180,E1 -13435.787,E2 -13435.787} C_VEL
LIN {X 0,Y 354.812,Z 286.103,A -85,B 0,C 180,E1 -13436.709,E2 -13436.709} C_VEL
LIN {X 0,Y 354.793,Z 286.105,A -85,B 0,C 180,E1 -13439.683,E2 -13439.683} C_VEL
LIN {X 0,Y 354.783,Z 286.103,A -85,B 0,C 180,E1 -13442.333,E2 -13442.333} C_VEL
LIN {X 0,Y 354.817,Z 286.101,A -85,B 0,C 180,E1 -13445.698,E2 -13445.698} C_VEL
LIN {X 0,Y 354.819,Z 286.104,A -85,B 0,C 180,E1 -13449.423,E2 -13449.423} C_VEL
LIN {X 0,Y 354.782,Z 286.106,A -85,B 0,C 180,E1 -13452.866,E2 -13452.866} C_VEL
LIN {X 0,Y 354.76,Z 286.107,A -85,B 0,C 180,E1 -13456.103,E2 -13456.103} C_VEL
LIN {X 0,Y 354.78,Z 286.101,A -85,B 0,C 180,E1 -13459.178,E2 -13459.178} C_VEL
LIN {X 0,Y 354.798,Z 286.094,A -85,B 0,C 180,E1 -13462.402,E2 -13462.402} C_VEL
LIN {X 0,Y 354.804,Z 286.099,A -85,B 0,C 180,E1 -13464.94,E2 -13464.94} C_VEL
LIN {X 0,Y 354.785,Z 286.1,A -85,B 0,C 180,E1 -13468.405,E2 -13468.405} C_VEL
LIN {X 0,Y 354.84,Z 286.093,A -85,B 0,C 180,E1 -13471.618,E2 -13471.618} C_VEL
LIN {X 0,Y 354.888,Z 286.089,A -85,B 0,C 180,E1 -13474.172,E2 -13474.172} C_VEL
LIN {X 0,Y 354.805,Z 286.092,A -85,B 0,C 180,E1 -13477.892,E2 -13477.892} C_VEL
LIN {X 0,Y 354.912,Z 286.088,A -85,B 0,C 180,E1 -13481.891,E2 -13481.891} C_VEL
LIN {X 0,Y 354.932,Z 286.078,A -85,B 0,C 180,E1 -13485.981,E2 -13485.981} C_VEL
LIN {X 0,Y 354.967,Z 286.073,A -85,B 0,C 180,E1 -13489.736,E2 -13489.736} C_VEL
LIN {X 0,Y 355.115,Z 286.06,A -85,B 0,C 180,E1 -13493.18,E2 -13493.18} C_VEL
LIN {X 0,Y 355.231,Z 286.039,A -85,B 0,C 180,E1 -13497.732,E2 -13497.732} C_VEL
LIN {X 0,Y 355.385,Z 286.024,A -85,B 0,C 180,E1 -13500,E2 -13500} C_VEL
LIN {X 0,Y 355.232,Z 286.036,A -85,B 0,C 180,E1 -13502.268,E2 -13502.268} C_VEL
LIN {X 0,Y 355.088,Z 286.063,A -85,B 0,C 180,E1 -13506.82,E2 -13506.82} C_VEL
LIN {X 0,Y 354.967,Z 286.079,A -85,B 0,C 180,E1 -13510.265,E2 -13510.265} C_VEL
LIN {X 0,Y 354.932,Z 286.085,A -85,B 0,C 180,E1 -13514.019,E2 -13514.019} C_VEL
LIN {X 0,Y 354.913,Z 286.09,A -85,B 0,C 180,E1 -13518.109,E2 -13518.109} C_VEL
LIN {X 0,Y 354.825,Z 286.102,A -85,B 0,C 180,E1 -13522.107,E2 -13522.107} C_VEL
LIN {X 0,Y 354.891,Z 286.093,A -85,B 0,C 180,E1 -13525.828,E2 -13525.828} C_VEL
LIN {X 0,Y 354.847,Z 286.095,A -85,B 0,C 180,E1 -13529.679,E2 -13529.679} C_VEL
LIN {X 0,Y 354.799,Z 286.104,A -85,B 0,C 180,E1 -13533.703,E2 -13533.703} C_VEL
LIN {X 0,Y 354.793,Z 286.105,A -85,B 0,C 180,E1 -13536.46,E2 -13536.46} C_VEL
LIN {X 0,Y 354.89,Z 286.126,A -85,B 0,C 180,E1 -13540.247,E2 -13540.247} C_VEL
LIN {X 0,Y 356.395,Z 294.026,A -85,B 0,C 180,E1 -13542.62,E2 -13542.62} C_VEL
LIN {X 0,Y 356.175,Z 298.978,A -85,B 0,C 180,E1 -13543.999,E2 -13543.999} C_VEL
LIN {X 0,Y 360.509,Z 320.822,A -85,B 0,C 180,E1 -13544.722,E2 -13544.722} C_VEL
LIN {X 0,Y 359.55,Z 376.408,A -85,B 0,C 180,E1 -13545.902,E2 -13545.902} C_VEL
LIN {X 0,Y 359.183,Z 387.11,A -85,B 0,C 180,E1 -13546.308,E2 -13546.308} C_VEL
LIN {X 0,Y 358.622,Z 398.571,A -85,B 0,C 180,E1 -13546.984,E2 -13546.984} C_VEL
LIN {X 0,Y 357.968,Z 407.986,A -85,B 0,C 180,E1 -13547.747,E2 -13547.747} C_VEL
LIN {X 0,Y 357.308,Z 415.892,A -85,B 0,C 180,E1 -13548.552,E2 -13548.552} C_VEL
LIN {X 0,Y 356.635,Z 423.026,A -85,B 0,C 180,E1 -13549.436,E2 -13549.436} C_VEL
LIN {X 0,Y 356.009,Z 429.164,A -85,B 0,C 180,E1 -13550.345,E2 -13550.345} C_VEL
LIN {X 0,Y 355.357,Z 435.456,A -85,B 0,C 180,E1 -13551.467,E2 -13551.467} C_VEL
LIN {X 0,Y 354.831,Z 440.933,A -85,B 0,C 180,E1 -13552.651,E2 -13552.651} C_VEL
LIN {X 0,Y 354.331,Z 446.08,A -85,B 0,C 180,E1 -13554.019,E2 -13554.019} C_VEL
LIN {X 0,Y 353.816,Z 450.534,A -85,B 0,C 180,E1 -13555.522,E2 -13555.522} C_VEL
LIN {X 0,Y 353.655,Z 452.983,A -85,B 0,C 180,E1 -13556.579,E2 -13556.579} C_VEL
LIN {X 0,Y 353.521,Z 454.838,A -85,B 0,C 180,E1 -13557.538,E2 -13557.538} C_VEL
LIN {X 0,Y 353.302,Z 456.676,A -85,B 0,C 180,E1 -13558.856,E2 -13558.856} C_VEL
LIN {X 0,Y 353.098,Z 457.792,A -85,B 0,C 180,E1 -13560.16,E2 -13560.16} C_VEL
LIN {X 0,Y 353.02,Z 458.228,A -85,B 0,C 180,E1 -13561.459,E2 -13561.459} C_VEL
LIN {X 0,Y 353.081,Z 457.57,A -85,B 0,C 180,E1 -13563.601,E2 -13563.601} C_VEL
LIN {X 0,Y 353.209,Z 455.754,A -85,B 0,C 180,E1 -13565.302,E2 -13565.302} C_VEL
LIN {X 0,Y 353.444,Z 453.662,A -85,B 0,C 180,E1 -13566.567,E2 -13566.567} C_VEL
LIN {X 0,Y 353.772,Z 449.245,A -85,B 0,C 180,E1 -13568.439,E2 -13568.439} C_VEL
LIN {X 0,Y 354.17,Z 444.311,A -85,B 0,C 180,E1 -13569.984,E2 -13569.984} C_VEL
LIN {X 0,Y 354.705,Z 437.903,A -85,B 0,C 180,E1 -13571.518,E2 -13571.518} C_VEL
LIN {X 0,Y 355.243,Z 431.51,A -85,B 0,C 180,E1 -13572.738,E2 -13572.738} C_VEL
LIN {X 0,Y 355.798,Z 424.761,A -85,B 0,C 180,E1 -13573.8,E2 -13573.8} C_VEL
LIN {X 0,Y 356.452,Z 416.843,A -85,B 0,C 180,E1 -13574.818,E2 -13574.818} C_VEL
LIN {X 0,Y 357.028,Z 409.306,A -85,B 0,C 180,E1 -13575.611,E2 -13575.611} C_VEL
LIN {X 0,Y 357.582,Z 400.451,A -85,B 0,C 180,E1 -13576.359,E2 -13576.359} C_VEL
LIN {X 0,Y 357.978,Z 391.4,A -85,B 0,C 180,E1 -13576.952,E2 -13576.952} C_VEL
LIN {X 0,Y 358.445,Z 380.277,A -85,B 0,C 180,E1 -13577.473,E2 -13577.473} C_VEL
LIN {X 0,Y 358.77,Z 365.377,A -85,B 0,C 180,E1 -13577.853,E2 -13577.853} C_VEL
LIN {X 0,Y 359.294,Z 320.298,A -85,B 0,C 180,E1 -13578.779,E2 -13578.779} C_VEL
LIN {X 0,Y 355.589,Z 299.08,A -85,B 0,C 180,E1 -13579.43,E2 -13579.43} C_VEL
LIN {X 0,Y 355.922,Z 292.394,A -85,B 0,C 180,E1 -13581.484,E2 -13581.484} C_VEL
LIN {X 0,Y 355.114,Z 286.066,A -85,B 0,C 180,E1 -13583.537,E2 -13583.537} C_VEL
LIN {X 0,Y 355.245,Z 286.048,A -85,B 0,C 180,E1 -13587.732,E2 -13587.732} C_VEL
LIN {X 0,Y 355.398,Z 286.029,A -85,B 0,C 180,E1 -13590,E2 -13590} C_VEL
LIN {X 0,Y 355.246,Z 286.046,A -85,B 0,C 180,E1 -13592.268,E2 -13592.268} C_VEL
LIN {X 0,Y 355.105,Z 286.061,A -85,B 0,C 180,E1 -13596.82,E2 -13596.82} C_VEL
LIN {X 0,Y 354.979,Z 286.083,A -85,B 0,C 180,E1 -13600.264,E2 -13600.264} C_VEL
LIN {X 0,Y 354.944,Z 286.083,A -85,B 0,C 180,E1 -13604.018,E2 -13604.018} C_VEL
LIN {X 0,Y 354.89,Z 286.089,A -85,B 0,C 180,E1 -13608.092,E2 -13608.092} C_VEL
LIN {X 0,Y 354.817,Z 286.097,A -85,B 0,C 180,E1 -13612.106,E2 -13612.106} C_VEL
LIN {X 0,Y 354.845,Z 286.093,A -85,B 0,C 180,E1 -13614.178,E2 -13614.178} C_VEL
LIN {X 0,Y 354.227,Z 286.177,A -85,B 0,C 180,E1 -13615.126,E2 -13615.126} C_VEL
LIN {X 0,Y 351.38,Z 286.538,A -85,B 0,C 180,E1 -13616.668,E2 -13616.668} C_VEL
LIN {X 0,Y 348.936,Z 286.841,A -85,B 0,C 180,E1 -13617.916,E2 -13617.916} C_VEL
LIN {X 0,Y 347.885,Z 286.966,A -85,B 0,C 180,E1 -13618.882,E2 -13618.882} C_VEL
LIN {X 0,Y 347.8,Z 286.974,A -85,B 0,C 180,E1 -13619.209,E2 -13619.209} C_VEL
LIN {X 0,Y 347.731,Z 286.985,A -85,B 0,C 180,E1 -13623.071,E2 -13623.071} C_VEL
LIN {X 0,Y 347.767,Z 286.974,A -85,B 0,C 180,E1 -13626.064,E2 -13626.064} C_VEL
LIN {X 0,Y 347.749,Z 286.978,A -85,B 0,C 180,E1 -13628.792,E2 -13628.792} C_VEL
LIN {X 0,Y 347.747,Z 286.979,A -85,B 0,C 180,E1 -13631.829,E2 -13631.829} C_VEL
LIN {X 0,Y 347.792,Z 286.973,A -85,B 0,C 180,E1 -13635.011,E2 -13635.011} C_VEL
LIN {X 0,Y 347.781,Z 286.973,A -85,B 0,C 180,E1 -13638.39,E2 -13638.39} C_VEL
LIN {X 0,Y 347.769,Z 286.978,A -85,B 0,C 180,E1 -13642.01,E2 -13642.01} C_VEL
LIN {X 0,Y 347.738,Z 286.981,A -85,B 0,C 180,E1 -13645.535,E2 -13645.535} C_VEL
LIN {X 0,Y 347.757,Z 286.978,A -85,B 0,C 180,E1 -13649.653,E2 -13649.653} C_VEL
LIN {X 0,Y 347.845,Z 286.965,A -85,B 0,C 180,E1 -13652.744,E2 -13652.744} C_VEL
LIN {X 0,Y 347.78,Z 286.978,A -85,B 0,C 180,E1 -13656.161,E2 -13656.161} C_VEL
LIN {X 0,Y 347.801,Z 286.972,A -85,B 0,C 180,E1 -13659.909,E2 -13659.909} C_VEL
LIN {X 0,Y 347.857,Z 286.968,A -85,B 0,C 180,E1 -13662.359,E2 -13662.359} C_VEL
LIN {X 0,Y 347.888,Z 286.96,A -85,B 0,C 180,E1 -13665.97,E2 -13665.97} C_VEL
LIN {X 0,Y 347.918,Z 286.956,A -85,B 0,C 180,E1 -13669.525,E2 -13669.525} C_VEL
LIN {X 0,Y 348.081,Z 286.94,A -85,B 0,C 180,E1 -13673.042,E2 -13673.042} C_VEL
LIN {X 0,Y 348.197,Z 286.921,A -85,B 0,C 180,E1 -13677.686,E2 -13677.686} C_VEL
LIN {X 0,Y 348.335,Z 286.903,A -85,B 0,C 180,E1 -13680,E2 -13680} C_VEL
LIN {X 0,Y 348.195,Z 286.921,A -85,B 0,C 180,E1 -13682.313,E2 -13682.313} C_VEL
LIN {X 0,Y 348.08,Z 286.938,A -85,B 0,C 180,E1 -13686.958,E2 -13686.958} C_VEL
LIN {X 0,Y 347.922,Z 286.955,A -85,B 0,C 180,E1 -13690.474,E2 -13690.474} C_VEL
LIN {X 0,Y 347.889,Z 286.96,A -85,B 0,C 180,E1 -13694.15,E2 -13694.15} C_VEL
LIN {X 0,Y 347.881,Z 286.961,A -85,B 0,C 180,E1 -13698.29,E2 -13698.29} C_VEL
LIN {X 0,Y 347.766,Z 286.978,A -85,B 0,C 180,E1 -13701.63,E2 -13701.63} C_VEL
LIN {X 0,Y 347.802,Z 286.97,A -85,B 0,C 180,E1 -13705.109,E2 -13705.109} C_VEL
LIN {X 0,Y 347.799,Z 286.973,A -85,B 0,C 180,E1 -13707.695,E2 -13707.695} C_VEL
LIN {X 0,Y 347.741,Z 286.982,A -85,B 0,C 180,E1 -13710.349,E2 -13710.349} C_VEL
LIN {X 0,Y 347.741,Z 286.981,A -85,B 0,C 180,E1 -13714.044,E2 -13714.044} C_VEL
LIN {X 0,Y 347.753,Z 286.976,A -85,B 0,C 180,E1 -13717.322,E2 -13717.322} C_VEL
LIN {X 0,Y 347.725,Z 286.983,A -85,B 0,C 180,E1 -13720.298,E2 -13720.298} C_VEL
LIN {X 0,Y 347.72,Z 286.98,A -85,B 0,C 180,E1 -13723.408,E2 -13723.408} C_VEL
LIN {X 0,Y 347.72,Z 286.986,A -85,B 0,C 180,E1 -13726.687,E2 -13726.687} C_VEL
LIN {X 0,Y 347.742,Z 286.978,A -85,B 0,C 180,E1 -13730.174,E2 -13730.174} C_VEL
LIN {X 0,Y 347.756,Z 286.979,A -85,B 0,C 180,E1 -13732.68,E2 -13732.68} C_VEL
LIN {X 0,Y 347.745,Z 286.977,A -85,B 0,C 180,E1 -13735.957,E2 -13735.957} C_VEL
LIN {X 0,Y 347.737,Z 286.98,A -85,B 0,C 180,E1 -13739.652,E2 -13739.652} C_VEL
LIN {X 0,Y 347.799,Z 287.037,A -85,B 0,C 180,E1 -13743.477,E2 -13743.477} C_VEL
LIN {X 0,Y 349.887,Z 298.478,A -85,B 0,C 180,E1 -13746.942,E2 -13746.942} C_VEL
LIN {X 0,Y 349.266,Z 306.049,A -85,B 0,C 180,E1 -13749.074,E2 -13749.074} C_VEL
LIN {X 0,Y 348.326,Z 317.7,A -85,B 0,C 180,E1 -13752.301,E2 -13752.301} C_VEL
LIN {X 0,Y 352.247,Z 347.256,A -85,B 0,C 180,E1 -13753.12,E2 -13753.12} C_VEL
LIN {X 0,Y 351.547,Z 395.263,A -85,B 0,C 180,E1 -13754.157,E2 -13754.157} C_VEL
LIN {X 0,Y 351.037,Z 406.378,A -85,B 0,C 180,E1 -13754.58,E2 -13754.58} C_VEL
LIN {X 0,Y 350.383,Z 416.706,A -85,B 0,C 180,E1 -13755.183,E2 -13755.183} C_VEL
LIN {X 0,Y 349.744,Z 427.218,A -85,B 0,C 180,E1 -13756.047,E2 -13756.047} C_VEL
LIN {X 0,Y 349.054,Z 435.48,A -85,B 0,C 180,E1 -13756.909,E2 -13756.909} C_VEL
LIN {X 0,Y 348.427,Z 443.321,A -85,B 0,C 180,E1 -13757.921,E2 -13757.921} C_VEL
LIN {X 0,Y 347.877,Z 449.799,A -85,B 0,C 180,E1 -13758.935,E2 -13758.935} C_VEL
LIN {X 0,Y 347.308,Z 455.965,A -85,B 0,C 180,E1 -13760.096,E2 -13760.096} C_VEL
LIN {X 0,Y 346.809,Z 462.262,A -85,B 0,C 180,E1 -13761.552,E2 -13761.552} C_VEL
LIN {X 0,Y 346.461,Z 467.252,A -85,B 0,C 180,E1 -13763.009,E2 -13763.009} C_VEL
LIN {X 0,Y 346.231,Z 471.728,A -85,B 0,C 180,E1 -13764.759,E2 -13764.759} C_VEL
LIN {X 0,Y 346.166,Z 474.843,A -85,B 0,C 180,E1 -13766.508,E2 -13766.508} C_VEL
LIN {X 0,Y 346.089,Z 476.28,A -85,B 0,C 180,E1 -13767.672,E2 -13767.672} C_VEL
LIN {X 0,Y 346.103,Z 477.212,A -85,B 0,C 180,E1 -13768.836,E2 -13768.836} C_VEL
LIN {X 0,Y 346.162,Z 477.545,A -85,B 0,C 180,E1 -13770,E2 -13770} C_VEL
LIN {X 0,Y 346.101,Z 477.377,A -85,B 0,C 180,E1 -13771.163,E2 -13771.163} C_VEL
LIN {X 0,Y 346.087,Z 476.744,A -85,B 0,C 180,E1 -13772.328,E2 -13772.328} C_VEL
LIN {X 0,Y 346.166,Z 475.637,A -85,B 0,C 180,E1 -13773.492,E2 -13773.492} C_VEL
LIN {X 0,Y 346.244,Z 472.866,A -85,B 0,C 180,E1 -13775.241,E2 -13775.241} C_VEL
LIN {X 0,Y 346.358,Z 470.531,A -85,B 0,C 180,E1 -13776.349,E2 -13776.349} C_VEL
LIN {X 0,Y 346.667,Z 467.265,A -85,B 0,C 180,E1 -13777.572,E2 -13777.572} C_VEL
LIN {X 0,Y 347.184,Z 461.147,A -85,B 0,C 180,E1 -13779.319,E2 -13779.319} C_VEL
LIN {X 0,Y 347.699,Z 456.1,A -85,B 0,C 180,E1 -13780.481,E2 -13780.481} C_VEL
LIN {X 0,Y 348.368,Z 450.029,A -85,B 0,C 180,E1 -13781.638,E2 -13781.638} C_VEL
LIN {X 0,Y 349.067,Z 442.651,A -85,B 0,C 180,E1 -13782.795,E2 -13782.795} C_VEL
LIN {X 0,Y 349.89,Z 434.762,A -85,B 0,C 180,E1 -13783.799,E2 -13783.799} C_VEL
LIN {X 0,Y 350.649,Z 426.443,A -85,B 0,C 180,E1 -13784.657,E2 -13784.657} C_VEL
LIN {X 0,Y 351.497,Z 415.855,A -85,B 0,C 180,E1 -13785.511,E2 -13785.511} C_VEL
LIN {X 0,Y 352.231,Z 404.436,A -85,B 0,C 180,E1 -13786.146,E2 -13786.146} C_VEL
LIN {X 0,Y 352.718,Z 394.266,A -85,B 0,C 180,E1 -13786.518,E2 -13786.518} C_VEL
LIN {X 0,Y 353.307,Z 345.656,A -85,B 0,C 180,E1 -13787.584,E2 -13787.584} C_VEL
LIN {X 0,Y 349.464,Z 320.605,A -85,B 0,C 180,E1 -13788.366,E2 -13788.366} C_VEL
LIN {X 0,Y 348.767,Z 316.736,A -85,B 0,C 180,E1 -13788.514,E2 -13788.514} C_VEL
LIN {X 0,Y 350.079,Z 301.866,A -85,B 0,C 180,E1 -13792.562,E2 -13792.562} C_VEL
LIN {X 0,Y 349.95,Z 297.92,A -85,B 0,C 180,E1 -13793.681,E2 -13793.681} C_VEL
LIN {X 0,Y 347.767,Z 286.979,A -85,B 0,C 180,E1 -13797.01,E2 -13797.01} C_VEL
LIN {X 0,Y 347.734,Z 286.987,A -85,B 0,C 180,E1 -13800.348,E2 -13800.348} C_VEL
LIN {X 0,Y 347.744,Z 286.98,A -85,B 0,C 180,E1 -13804.043,E2 -13804.043} C_VEL
LIN {X 0,Y 347.756,Z 286.983,A -85,B 0,C 180,E1 -13807.32,E2 -13807.32} C_VEL
LIN {X 0,Y 347.726,Z 286.987,A -85,B 0,C 180,E1 -13810.296,E2 -13810.296} C_VEL
LIN {X 0,Y 347.717,Z 286.992,A -85,B 0,C 180,E1 -13813.407,E2 -13813.407} C_VEL
LIN {X 0,Y 347.718,Z 286.985,A -85,B 0,C 180,E1 -13816.686,E2 -13816.686} C_VEL
LIN {X 0,Y 347.74,Z 286.98,A -85,B 0,C 180,E1 -13820.172,E2 -13820.172} C_VEL
LIN {X 0,Y 347.753,Z 286.972,A -85,B 0,C 180,E1 -13822.678,E2 -13822.678} C_VEL
LIN {X 0,Y 347.74,Z 286.978,A -85,B 0,C 180,E1 -13825.956,E2 -13825.956} C_VEL
LIN {X 0,Y 347.755,Z 286.979,A -85,B 0,C 180,E1 -13829.653,E2 -13829.653} C_VEL
LIN {X 0,Y 347.842,Z 286.957,A -85,B 0,C 180,E1 -13832.745,E2 -13832.745} C_VEL
LIN {X 0,Y 347.775,Z 286.975,A -85,B 0,C 180,E1 -13836.161,E2 -13836.161} C_VEL
LIN {X 0,Y 347.795,Z 286.969,A -85,B 0,C 180,E1 -13839.908,E2 -13839.908} C_VEL
LIN {X 0,Y 347.856,Z 286.965,A -85,B 0,C 180,E1 -13842.359,E2 -13842.359} C_VEL
LIN {X 0,Y 347.888,Z 286.956,A -85,B 0,C 180,E1 -13845.971,E2 -13845.971} C_VEL
LIN {X 0,Y 347.918,Z 286.95,A -85,B 0,C 180,E1 -13849.525,E2 -13849.525} C_VEL
LIN {X 0,Y 348.081,Z 286.937,A -85,B 0,C 180,E1 -13853.042,E2 -13853.042} C_VEL
LIN {X 0,Y 348.194,Z 286.916,A -85,B 0,C 180,E1 -13857.687,E2 -13857.687} C_VEL
LIN {X 0,Y 348.334,Z 286.903,A -85,B 0,C 180,E1 -13860,E2 -13860} C_VEL
LIN {X 0,Y 348.194,Z 286.912,A -85,B 0,C 180,E1 -13862.314,E2 -13862.314} C_VEL
LIN {X 0,Y 348.056,Z 286.937,A -85,B 0,C 180,E1 -13866.959,E2 -13866.959} C_VEL
LIN {X 0,Y 347.918,Z 286.957,A -85,B 0,C 180,E1 -13870.475,E2 -13870.475} C_VEL
LIN {X 0,Y 347.889,Z 286.962,A -85,B 0,C 180,E1 -13874.15,E2 -13874.15} C_VEL
LIN {X 0,Y 347.881,Z 286.965,A -85,B 0,C 180,E1 -13878.291,E2 -13878.291} C_VEL
LIN {X 0,Y 347.78,Z 286.979,A -85,B 0,C 180,E1 -13881.636,E2 -13881.636} C_VEL
LIN {X 0,Y 347.804,Z 286.974,A -85,B 0,C 180,E1 -13885.109,E2 -13885.109} C_VEL
LIN {X 0,Y 347.804,Z 286.974,A -85,B 0,C 180,E1 -13887.695,E2 -13887.695} C_VEL
LIN {X 0,Y 347.757,Z 286.979,A -85,B 0,C 180,E1 -13890.347,E2 -13890.347} C_VEL
LIN {X 0,Y 347.737,Z 286.979,A -85,B 0,C 180,E1 -13894.465,E2 -13894.465} C_VEL
LIN {X 0,Y 347.77,Z 286.98,A -85,B 0,C 180,E1 -13897.99,E2 -13897.99} C_VEL
LIN {X 0,Y 347.82,Z 287.061,A -85,B 0,C 180,E1 -13899.943,E2 -13899.943} C_VEL
LIN {X 0,Y 349.376,Z 294.955,A -85,B 0,C 180,E1 -13902.376,E2 -13902.376} C_VEL
LIN {X 0,Y 349.34,Z 299.307,A -85,B 0,C 180,E1 -13903.59,E2 -13903.59} C_VEL
LIN {X 0,Y 353.738,Z 321.45,A -85,B 0,C 180,E1 -13904.35,E2 -13904.35} C_VEL
LIN {X 0,Y 352.835,Z 376.19,A -85,B 0,C 180,E1 -13905.538,E2 -13905.538} C_VEL
LIN {X 0,Y 352.437,Z 386.498,A -85,B 0,C 180,E1 -13905.926,E2 -13905.926} C_VEL
LIN {X 0,Y 351.858,Z 398.627,A -85,B 0,C 180,E1 -13906.64,E2 -13906.64} C_VEL
LIN {X 0,Y 351.122,Z 408.446,A -85,B 0,C 180,E1 -13907.452,E2 -13907.452} C_VEL
LIN {X 0,Y 350.433,Z 416.371,A -85,B 0,C 180,E1 -13908.28,E2 -13908.28} C_VEL
LIN {X 0,Y 349.696,Z 423.746,A -85,B 0,C 180,E1 -13909.222,E2 -13909.222} C_VEL
LIN {X 0,Y 348.98,Z 430.421,A -85,B 0,C 180,E1 -13910.254,E2 -13910.254} C_VEL
LIN {X 0,Y 348.372,Z 436.014,A -85,B 0,C 180,E1 -13911.291,E2 -13911.291} C_VEL
LIN {X 0,Y 347.932,Z 440.69,A -85,B 0,C 180,E1 -13912.315,E2 -13912.315} C_VEL
LIN {X 0,Y 347.342,Z 445.939,A -85,B 0,C 180,E1 -13913.715,E2 -13913.715} C_VEL
LIN {X 0,Y 347.034,Z 449.162,A -85,B 0,C 180,E1 -13914.749,E2 -13914.749} C_VEL
LIN {X 0,Y 346.55,Z 453.907,A -85,B 0,C 180,E1 -13916.802,E2 -13916.802} C_VEL
LIN {X 0,Y 346.263,Z 456.518,A -85,B 0,C 180,E1 -13918.481,E2 -13918.481} C_VEL
LIN {X 0,Y 346.083,Z 457.504,A -85,B 0,C 180,E1 -13919.492,E2 -13919.492} C_VEL
LIN {X 0,Y 345.939,Z 458.285,A -85,B 0,C 180,E1 -13920.877,E2 -13920.877} C_VEL
LIN {X 0,Y 345.91,Z 458.394,A -85,B 0,C 180,E1 -13922.142,E2 -13922.142} C_VEL
LIN {X 0,Y 345.99,Z 457.886,A -85,B 0,C 180,E1 -13923.457,E2 -13923.457} C_VEL
LIN {X 0,Y 346.074,Z 456.749,A -85,B 0,C 180,E1 -13924.758,E2 -13924.758} C_VEL
LIN {X 0,Y 346.25,Z 454.94,A -85,B 0,C 180,E1 -13926.05,E2 -13926.05} C_VEL
LIN {X 0,Y 346.603,Z 450.928,A -85,B 0,C 180,E1 -13927.969,E2 -13927.969} C_VEL
LIN {X 0,Y 346.895,Z 447.102,A -85,B 0,C 180,E1 -13929.327,E2 -13929.327} C_VEL
LIN {X 0,Y 347.357,Z 441.791,A -85,B 0,C 180,E1 -13930.806,E2 -13930.806} C_VEL
LIN {X 0,Y 347.841,Z 436.118,A -85,B 0,C 180,E1 -13932.078,E2 -13932.078} C_VEL
LIN {X 0,Y 348.458,Z 429.462,A -85,B 0,C 180,E1 -13933.298,E2 -13933.298} C_VEL
LIN {X 0,Y 349.18,Z 421.169,A -85,B 0,C 180,E1 -13934.533,E2 -13934.533} C_VEL
LIN {X 0,Y 349.886,Z 412.019,A -85,B 0,C 180,E1 -13935.608,E2 -13935.608} C_VEL
LIN {X 0,Y 350.52,Z 403.704,A -85,B 0,C 180,E1 -13936.374,E2 -13936.374} C_VEL
LIN {X 0,Y 350.948,Z 394.291,A -85,B 0,C 180,E1 -13937.054,E2 -13937.054} C_VEL
LIN {X 0,Y 351.37,Z 384.505,A -85,B 0,C 180,E1 -13937.573,E2 -13937.573} C_VEL
LIN {X 0,Y 351.702,Z 375.152,A -85,B 0,C 180,E1 -13937.907,E2 -13937.907} C_VEL
LIN {X 0,Y 352.376,Z 320.632,A -85,B 0,C 180,E1 -13939.079,E2 -13939.079} C_VEL
LIN {X 0,Y 348.622,Z 299.345,A -85,B 0,C 180,E1 -13939.73,E2 -13939.73} C_VEL
LIN {X 0,Y 348.946,Z 293.691,A -85,B 0,C 180,E1 -13941.495,E2 -13941.495} C_VEL
LIN {X 0,Y 348.1,Z 286.939,A -85,B 0,C 180,E1 -13943.77,E2 -13943.77} C_VEL
LIN {X 0,Y 348.208,Z 286.924,A -85,B 0,C 180,E1 -13947.687,E2 -13947.687} C_VEL
LIN {X 0,Y 348.347,Z 286.908,A -85,B 0,C 180,E1 -13950,E2 -13950} C_VEL
LIN {X 0,Y 348.208,Z 286.922,A -85,B 0,C 180,E1 -13952.313,E2 -13952.313} C_VEL
LIN {X 0,Y 348.072,Z 286.936,A -85,B 0,C 180,E1 -13956.958,E2 -13956.958} C_VEL
LIN {X 0,Y 347.93,Z 286.958,A -85,B 0,C 180,E1 -13960.474,E2 -13960.474} C_VEL
LIN {X 0,Y 347.9,Z 286.961,A -85,B 0,C 180,E1 -13964.149,E2 -13964.149} C_VEL
LIN {X 0,Y 347.829,Z 286.97,A -85,B 0,C 180,E1 -13968.258,E2 -13968.258} C_VEL
LIN {X 0,Y 347.768,Z 286.974,A -85,B 0,C 180,E1 -13971.626,E2 -13971.626} C_VEL
LIN {X 0,Y 347.811,Z 286.972,A -85,B 0,C 180,E1 -13975.108,E2 -13975.108} C_VEL
LIN {X 0,Y 347.809,Z 286.969,A -85,B 0,C 180,E1 -13977.693,E2 -13977.693} C_VEL
LIN {X 0,Y 347.8,Z 286.974,A -85,B 0,C 180,E1 -13979.209,E2 -13979.209} C_VEL
LIN {X 0,Y 347.118,Z 287.056,A -85,B 0,C 180,E1 -13980.176,E2 -13980.176} C_VEL
LIN {X 0,Y 344.21,Z 287.418,A -85,B 0,C 180,E1 -13981.747,E2 -13981.747} C_VEL
LIN {X 0,Y 341.777,Z 287.726,A -85,B 0,C 180,E1 -13983.019,E2 -13983.019} C_VEL
LIN {X 0,Y 340.775,Z 287.846,A -85,B 0,C 180,E1 -13984.004,E2 -13984.004} C_VEL
LIN {X 0,Y 340.715,Z 287.853,A -85,B 0,C 180,E1 -13984.337,E2 -13984.337} C_VEL
LIN {X 0,Y 340.73,Z 287.851,A -85,B 0,C 180,E1 -13988.226,E2 -13988.226} C_VEL
LIN {X 0,Y 340.696,Z 287.856,A -85,B 0,C 180,E1 -13992.045,E2 -13992.045} C_VEL
LIN {X 0,Y 340.732,Z 287.857,A -85,B 0,C 180,E1 -13995.469,E2 -13995.469} C_VEL
LIN {X 0,Y 340.721,Z 287.852,A -85,B 0,C 180,E1 -13998.695,E2 -13998.695} C_VEL
LIN {X 0,Y 340.73,Z 287.857,A -85,B 0,C 180,E1 -14001.772,E2 -14001.772} C_VEL
LIN {X 0,Y 340.716,Z 287.856,A -85,B 0,C 180,E1 -14005.595,E2 -14005.595} C_VEL
LIN {X 0,Y 340.697,Z 287.855,A -85,B 0,C 180,E1 -14008.955,E2 -14008.955} C_VEL
LIN {X 0,Y 340.772,Z 287.848,A -85,B 0,C 180,E1 -14012.473,E2 -14012.473} C_VEL
LIN {X 0,Y 340.748,Z 287.85,A -85,B 0,C 180,E1 -14015.638,E2 -14015.638} C_VEL
LIN {X 0,Y 340.734,Z 287.85,A -85,B 0,C 180,E1 -14019.473,E2 -14019.473} C_VEL
LIN {X 0,Y 340.848,Z 287.838,A -85,B 0,C 180,E1 -14021.984,E2 -14021.984} C_VEL
LIN {X 0,Y 340.86,Z 287.834,A -85,B 0,C 180,E1 -14025.705,E2 -14025.705} C_VEL
LIN {X 0,Y 340.861,Z 287.836,A -85,B 0,C 180,E1 -14029.306,E2 -14029.306} C_VEL
LIN {X 0,Y 341.049,Z 287.817,A -85,B 0,C 180,E1 -14032.898,E2 -14032.898} C_VEL
LIN {X 0,Y 341.158,Z 287.798,A -85,B 0,C 180,E1 -14037.639,E2 -14037.639} C_VEL
LIN {X 0,Y 341.285,Z 287.782,A -85,B 0,C 180,E1 -14040,E2 -14040} C_VEL
LIN {X 0,Y 341.157,Z 287.798,A -85,B 0,C 180,E1 -14042.361,E2 -14042.361} C_VEL
LIN {X 0,Y 341.048,Z 287.815,A -85,B 0,C 180,E1 -14047.102,E2 -14047.102} C_VEL
LIN {X 0,Y 340.864,Z 287.834,A -85,B 0,C 180,E1 -14050.694,E2 -14050.694} C_VEL
LIN {X 0,Y 340.854,Z 287.836,A -85,B 0,C 180,E1 -14054.325,E2 -14054.325} C_VEL
LIN {X 0,Y 340.827,Z 287.839,A -85,B 0,C 180,E1 -14058.466,E2 -14058.466} C_VEL
LIN {X 0,Y 340.712,Z 287.859,A -85,B 0,C 180,E1 -14061.843,E2 -14061.843} C_VEL
LIN {X 0,Y 340.763,Z 287.85,A -85,B 0,C 180,E1 -14065.665,E2 -14065.665} C_VEL
LIN {X 0,Y 340.72,Z 287.856,A -85,B 0,C 180,E1 -14068.321,E2 -14068.321} C_VEL
LIN {X 0,Y 340.689,Z 287.856,A -85,B 0,C 180,E1 -14071.045,E2 -14071.045} C_VEL
LIN {X 0,Y 340.71,Z 287.853,A -85,B 0,C 180,E1 -14075.28,E2 -14075.28} C_VEL
LIN {X 0,Y 340.702,Z 287.86,A -85,B 0,C 180,E1 -14078.387,E2 -14078.387} C_VEL
LIN {X 0,Y 340.692,Z 287.857,A -85,B 0,C 180,E1 -14082.046,E2 -14082.046} C_VEL
LIN {X 0,Y 340.676,Z 287.858,A -85,B 0,C 180,E1 -14085.462,E2 -14085.462} C_VEL
LIN {X 0,Y 340.68,Z 287.862,A -85,B 0,C 180,E1 -14088.691,E2 -14088.691} C_VEL
LIN {X 0,Y 340.728,Z 287.851,A -85,B 0,C 180,E1 -14091.773,E2 -14091.773} C_VEL
LIN {X 0,Y 340.719,Z 287.854,A -85,B 0,C 180,E1 -14095.596,E2 -14095.596} C_VEL
LIN {X 0,Y 340.691,Z 287.86,A -85,B 0,C 180,E1 -14098.956,E2 -14098.956} C_VEL
LIN {X 0,Y 340.754,Z 287.854,A -85,B 0,C 180,E1 -14103.182,E2 -14103.182} C_VEL
LIN {X 0,Y 342.661,Z 298.126,A -85,B 0,C 180,E1 -14106.426,E2 -14106.426} C_VEL
LIN {X 0,Y 342.856,Z 301.007,A -85,B 0,C 180,E1 -14107.283,E2 -14107.283} C_VEL
LIN {X 0,Y 341.606,Z 314.555,A -85,B 0,C 180,E1 -14111.151,E2 -14111.151} C_VEL
LIN {X 0,Y 341.365,Z 317.473,A -85,B 0,C 180,E1 -14111.971,E2 -14111.971} C_VEL
LIN {X 0,Y 345.38,Z 348.179,A -85,B 0,C 180,E1 -14112.84,E2 -14112.84} C_VEL
LIN {X 0,Y 344.672,Z 394.899,A -85,B 0,C 180,E1 -14113.87,E2 -14113.87} C_VEL
LIN {X 0,Y 344.206,Z 404.418,A -85,B 0,C 180,E1 -14114.228,E2 -14114.228} C_VEL
LIN {X 0,Y 343.532,Z 415.943,A -85,B 0,C 180,E1 -14114.881,E2 -14114.881} C_VEL
LIN {X 0,Y 342.839,Z 426.594,A -85,B 0,C 180,E1 -14115.76,E2 -14115.76} C_VEL
LIN {X 0,Y 342.143,Z 434.935,A -85,B 0,C 180,E1 -14116.639,E2 -14116.639} C_VEL
LIN {X 0,Y 341.461,Z 442.834,A -85,B 0,C 180,E1 -14117.67,E2 -14117.67} C_VEL
LIN {X 0,Y 340.903,Z 449.363,A -85,B 0,C 180,E1 -14118.706,E2 -14118.706} C_VEL
LIN {X 0,Y 340.288,Z 455.571,A -85,B 0,C 180,E1 -14119.89,E2 -14119.89} C_VEL
LIN {X 0,Y 339.779,Z 461.905,A -85,B 0,C 180,E1 -14121.376,E2 -14121.376} C_VEL
LIN {X 0,Y 339.408,Z 466.932,A -85,B 0,C 180,E1 -14122.863,E2 -14122.863} C_VEL
LIN {X 0,Y 339.156,Z 471.068,A -85,B 0,C 180,E1 -14124.457,E2 -14124.457} C_VEL
LIN {X 0,Y 339.093,Z 474.594,A -85,B 0,C 180,E1 -14126.435,E2 -14126.435} C_VEL
LIN {X 0,Y 339.004,Z 476.053,A -85,B 0,C 180,E1 -14127.624,E2 -14127.624} C_VEL
LIN {X 0,Y 339.006,Z 476.994,A -85,B 0,C 180,E1 -14128.812,E2 -14128.812} C_VEL
LIN {X 0,Y 339.065,Z 477.338,A -85,B 0,C 180,E1 -14130,E2 -14130} C_VEL
LIN {X 0,Y 339.004,Z 477.19,A -85,B 0,C 180,E1 -14131.188,E2 -14131.188} C_VEL
LIN {X 0,Y 339.002,Z 476.578,A -85,B 0,C 180,E1 -14132.376,E2 -14132.376} C_VEL
LIN {X 0,Y 339.093,Z 475.491,A -85,B 0,C 180,E1 -14133.565,E2 -14133.565} C_VEL
LIN {X 0,Y 339.151,Z 473.835,A -85,B 0,C 180,E1 -14134.754,E2 -14134.754} C_VEL
LIN {X 0,Y 339.314,Z 470.428,A -85,B 0,C 180,E1 -14136.481,E2 -14136.481} C_VEL
LIN {X 0,Y 339.596,Z 467.174,A -85,B 0,C 180,E1 -14137.731,E2 -14137.731} C_VEL
LIN {X 0,Y 340.18,Z 461.095,A -85,B 0,C 180,E1 -14139.513,E2 -14139.513} C_VEL
LIN {X 0,Y 340.714,Z 456.077,A -85,B 0,C 180,E1 -14140.698,E2 -14140.698} C_VEL
LIN {X 0,Y 341.419,Z 450.039,A -85,B 0,C 180,E1 -14141.879,E2 -14141.879} C_VEL
LIN {X 0,Y 342.141,Z 442.701,A -85,B 0,C 180,E1 -14143.059,E2 -14143.059} C_VEL
LIN {X 0,Y 343.011,Z 434.862,A -85,B 0,C 180,E1 -14144.081,E2 -14144.081} C_VEL
LIN {X 0,Y 343.803,Z 426.607,A -85,B 0,C 180,E1 -14144.956,E2 -14144.956} C_VEL
LIN {X 0,Y 344.687,Z 416.138,A -85,B 0,C 180,E1 -14145.825,E2 -14145.825} C_VEL
LIN {X 0,Y 345.484,Z 404.221,A -85,B 0,C 180,E1 -14146.508,E2 -14146.508} C_VEL
LIN {X 0,Y 345.944,Z 395.117,A -85,B 0,C 180,E1 -14146.857,E2 -14146.857} C_VEL
LIN {X 0,Y 346.61,Z 358.983,A -85,B 0,C 180,E1 -14147.673,E2 -14147.673} C_VEL
LIN {X 0,Y 346.535,Z 345.68,A -85,B 0,C 180,E1 -14147.977,E2 -14147.977} C_VEL
LIN {X 0,Y 342.908,Z 322.218,A -85,B 0,C 180,E1 -14148.736,E2 -14148.736} C_VEL
LIN {X 0,Y 341.868,Z 316.56,A -85,B 0,C 180,E1 -14148.939,E2 -14148.939} C_VEL
LIN {X 0,Y 343.165,Z 302.318,A -85,B 0,C 180,E1 -14152.899,E2 -14152.899} C_VEL
LIN {X 0,Y 342.752,Z 297.885,A -85,B 0,C 180,E1 -14154.21,E2 -14154.21} C_VEL
LIN {X 0,Y 340.718,Z 287.857,A -85,B 0,C 180,E1 -14157.383,E2 -14157.383} C_VEL
LIN {X 0,Y 340.689,Z 287.858,A -85,B 0,C 180,E1 -14161.044,E2 -14161.044} C_VEL
LIN {X 0,Y 340.713,Z 287.858,A -85,B 0,C 180,E1 -14165.278,E2 -14165.278} C_VEL
LIN {X 0,Y 340.704,Z 287.862,A -85,B 0,C 180,E1 -14168.385,E2 -14168.385} C_VEL
LIN {X 0,Y 340.693,Z 287.859,A -85,B 0,C 180,E1 -14172.044,E2 -14172.044} C_VEL
LIN {X 0,Y 340.645,Z 287.865,A -85,B 0,C 180,E1 -14176.226,E2 -14176.226} C_VEL
LIN {X 0,Y 340.681,Z 287.861,A -85,B 0,C 180,E1 -14179.752,E2 -14179.752} C_VEL
LIN {X 0,Y 340.697,Z 287.852,A -85,B 0,C 180,E1 -14183.258,E2 -14183.258} C_VEL
LIN {X 0,Y 340.684,Z 287.855,A -85,B 0,C 180,E1 -14186.153,E2 -14186.153} C_VEL
LIN {X 0,Y 340.766,Z 287.848,A -85,B 0,C 180,E1 -14190.332,E2 -14190.332} C_VEL
LIN {X 0,Y 340.795,Z 287.834,A -85,B 0,C 180,E1 -14193.019,E2 -14193.019} C_VEL
LIN {X 0,Y 340.745,Z 287.852,A -85,B 0,C 180,E1 -14195.638,E2 -14195.638} C_VEL
LIN {X 0,Y 340.723,Z 287.847,A -85,B 0,C 180,E1 -14199.473,E2 -14199.473} C_VEL
LIN {X 0,Y 340.848,Z 287.841,A -85,B 0,C 180,E1 -14201.984,E2 -14201.984} C_VEL
LIN {X 0,Y 340.86,Z 287.829,A -85,B 0,C 180,E1 -14205.705,E2 -14205.705} C_VEL
LIN {X 0,Y 340.86,Z 287.83,A -85,B 0,C 180,E1 -14209.306,E2 -14209.306} C_VEL
LIN {X 0,Y 341.049,Z 287.814,A -85,B 0,C 180,E1 -14212.898,E2 -14212.898} C_VEL
LIN {X 0,Y 341.156,Z 287.793,A -85,B 0,C 180,E1 -14217.639,E2 -14217.639} C_VEL
LIN {X 0,Y 341.285,Z 287.781,A -85,B 0,C 180,E1 -14220,E2 -14220} C_VEL
LIN {X 0,Y 341.156,Z 287.789,A -85,B 0,C 180,E1 -14222.361,E2 -14222.361} C_VEL
LIN {X 0,Y 341.005,Z 287.813,A -85,B 0,C 180,E1 -14227.103,E2 -14227.103} C_VEL
LIN {X 0,Y 340.86,Z 287.837,A -85,B 0,C 180,E1 -14230.694,E2 -14230.694} C_VEL
LIN {X 0,Y 340.854,Z 287.838,A -85,B 0,C 180,E1 -14234.325,E2 -14234.325} C_VEL
LIN {X 0,Y 340.828,Z 287.843,A -85,B 0,C 180,E1 -14238.467,E2 -14238.467} C_VEL
LIN {X 0,Y 340.745,Z 287.858,A -85,B 0,C 180,E1 -14241.858,E2 -14241.858} C_VEL
LIN {X 0,Y 340.764,Z 287.855,A -85,B 0,C 180,E1 -14245.665,E2 -14245.665} C_VEL
LIN {X 0,Y 340.734,Z 287.853,A -85,B 0,C 180,E1 -14248.32,E2 -14248.32} C_VEL
LIN {X 0,Y 340.697,Z 287.857,A -85,B 0,C 180,E1 -14251.045,E2 -14251.045} C_VEL
LIN {X 0,Y 340.712,Z 287.852,A -85,B 0,C 180,E1 -14255.28,E2 -14255.28} C_VEL
LIN {X 0,Y 340.729,Z 287.855,A -85,B 0,C 180,E1 -14259.381,E2 -14259.381} C_VEL
LIN {X 0,Y 340.787,Z 288.063,A -85,B 0,C 180,E1 -14259.648,E2 -14259.648} C_VEL
LIN {X 0,Y 342.475,Z 296.712,A -85,B 0,C 180,E1 -14262.376,E2 -14262.376} C_VEL
LIN {X 0,Y 342.484,Z 299.538,A -85,B 0,C 180,E1 -14263.158,E2 -14263.158} C_VEL
LIN {X 0,Y 347.083,Z 322.224,A -85,B 0,C 180,E1 -14263.968,E2 -14263.968} C_VEL
LIN {X 0,Y 346.119,Z 376.143,A -85,B 0,C 180,E1 -14265.161,E2 -14265.161} C_VEL
LIN {X 0,Y 345.758,Z 385.547,A -85,B 0,C 180,E1 -14265.513,E2 -14265.513} C_VEL
LIN {X 0,Y 345.231,Z 396.34,A -85,B 0,C 180,E1 -14266.116,E2 -14266.116} C_VEL
LIN {X 0,Y 344.453,Z 407.078,A -85,B 0,C 180,E1 -14266.967,E2 -14266.967} C_VEL
LIN {X 0,Y 343.611,Z 416.429,A -85,B 0,C 180,E1 -14267.946,E2 -14267.946} C_VEL
LIN {X 0,Y 342.911,Z 423.249,A -85,B 0,C 180,E1 -14268.823,E2 -14268.823} C_VEL
LIN {X 0,Y 342.252,Z 429.24,A -85,B 0,C 180,E1 -14269.737,E2 -14269.737} C_VEL
LIN {X 0,Y 341.451,Z 436.048,A -85,B 0,C 180,E1 -14270.998,E2 -14270.998} C_VEL
LIN {X 0,Y 340.914,Z 441.269,A -85,B 0,C 180,E1 -14272.173,E2 -14272.173} C_VEL
LIN {X 0,Y 340.453,Z 445.25,A -85,B 0,C 180,E1 -14273.228,E2 -14273.228} C_VEL
LIN {X 0,Y 339.993,Z 449.554,A -85,B 0,C 180,E1 -14274.636,E2 -14274.636} C_VEL
LIN {X 0,Y 339.561,Z 452.904,A -85,B 0,C 180,E1 -14276.026,E2 -14276.026} C_VEL
LIN {X 0,Y 339.396,Z 455.445,A -85,B 0,C 180,E1 -14277.427,E2 -14277.427} C_VEL
LIN {X 0,Y 339.102,Z 457.216,A -85,B 0,C 180,E1 -14278.794,E2 -14278.794} C_VEL
LIN {X 0,Y 338.883,Z 458.422,A -85,B 0,C 180,E1 -14280.579,E2 -14280.579} C_VEL
LIN {X 0,Y 338.812,Z 458.661,A -85,B 0,C 180,E1 -14281.505,E2 -14281.505} C_VEL
LIN {X 0,Y 338.853,Z 458.301,A -85,B 0,C 180,E1 -14283.106,E2 -14283.106} C_VEL
LIN {X 0,Y 338.919,Z 457.474,A -85,B 0,C 180,E1 -14284.186,E2 -14284.186} C_VEL
LIN {X 0,Y 339.095,Z 455.581,A -85,B 0,C 180,E1 -14285.774,E2 -14285.774} C_VEL
LIN {X 0,Y 339.415,Z 452.496,A -85,B 0,C 180,E1 -14287.477,E2 -14287.477} C_VEL
LIN {X 0,Y 339.834,Z 447.363,A -85,B 0,C 180,E1 -14289.417,E2 -14289.417} C_VEL
LIN {X 0,Y 340.223,Z 442.966,A -85,B 0,C 180,E1 -14290.701,E2 -14290.701} C_VEL
LIN {X 0,Y 340.709,Z 437.607,A -85,B 0,C 180,E1 -14291.977,E2 -14291.977} C_VEL
LIN {X 0,Y 341.335,Z 431.062,A -85,B 0,C 180,E1 -14293.247,E2 -14293.247} C_VEL
LIN {X 0,Y 341.942,Z 424.148,A -85,B 0,C 180,E1 -14294.35,E2 -14294.35} C_VEL
LIN {X 0,Y 342.619,Z 416.393,A -85,B 0,C 180,E1 -14295.365,E2 -14295.365} C_VEL
LIN {X 0,Y 343.277,Z 408.226,A -85,B 0,C 180,E1 -14296.232,E2 -14296.232} C_VEL
LIN {X 0,Y 343.919,Z 398.04,A -85,B 0,C 180,E1 -14297.085,E2 -14297.085} C_VEL
LIN {X 0,Y 344.445,Z 386.812,A -85,B 0,C 180,E1 -14297.753,E2 -14297.753} C_VEL
LIN {X 0,Y 344.787,Z 377.114,A -85,B 0,C 180,E1 -14298.138,E2 -14298.138} C_VEL
LIN {X 0,Y 345.291,Z 347.918,A -85,B 0,C 180,E1 -14298.799,E2 -14298.799} C_VEL
LIN {X 0,Y 345.516,Z 321.382,A -85,B 0,C 180,E1 -14299.374,E2 -14299.374} C_VEL
LIN {X 0,Y 341.666,Z 299.462,A -85,B 0,C 180,E1 -14300.081,E2 -14300.081} C_VEL
LIN {X 0,Y 341.901,Z 294.298,A -85,B 0,C 180,E1 -14301.727,E2 -14301.727} C_VEL
LIN {X 0,Y 341.06,Z 287.815,A -85,B 0,C 180,E1 -14303.938,E2 -14303.938} C_VEL
LIN {X 0,Y 341.169,Z 287.8,A -85,B 0,C 180,E1 -14307.639,E2 -14307.639} C_VEL
LIN {X 0,Y 341.297,Z 287.786,A -85,B 0,C 180,E1 -14310,E2 -14310} C_VEL
LIN {X 0,Y 341.17,Z 287.799,A -85,B 0,C 180,E1 -14312.361,E2 -14312.361} C_VEL
LIN {X 0,Y 341.02,Z 287.815,A -85,B 0,C 180,E1 -14317.103,E2 -14317.103} C_VEL
LIN {X 0,Y 340.872,Z 287.835,A -85,B 0,C 180,E1 -14320.693,E2 -14320.693} C_VEL
LIN {X 0,Y 340.864,Z 287.84,A -85,B 0,C 180,E1 -14324.324,E2 -14324.324} C_VEL
LIN {X 0,Y 340.786,Z 287.849,A -85,B 0,C 180,E1 -14328.44,E2 -14328.44} C_VEL
LIN {X 0,Y 340.718,Z 287.852,A -85,B 0,C 180,E1 -14331.841,E2 -14331.841} C_VEL
LIN {X 0,Y 340.771,Z 287.846,A -85,B 0,C 180,E1 -14335.664,E2 -14335.664} C_VEL
LIN {X 0,Y 340.741,Z 287.847,A -85,B 0,C 180,E1 -14339.219,E2 -14339.219} C_VEL
LIN {X 0,Y 340.684,Z 287.857,A -85,B 0,C 180,E1 -14342.435,E2 -14342.435} C_VEL
LIN {X 0,Y 340.715,Z 287.853,A -85,B 0,C 180,E1 -14344.337,E2 -14344.337} C_VEL
LIN {X 0,Y 340.104,Z 287.934,A -85,B 0,C 180,E1 -14345.324,E2 -14345.324} C_VEL
LIN {X 0,Y 337.253,Z 288.293,A -85,B 0,C 180,E1 -14346.929,E2 -14346.929} C_VEL
LIN {X 0,Y 334.79,Z 288.599,A -85,B 0,C 180,E1 -14348.229,E2 -14348.229} C_VEL
LIN {X 0,Y 333.716,Z 288.73,A -85,B 0,C 180,E1 -14349.235,E2 -14349.235} C_VEL
LIN {X 0,Y 333.622,Z 288.738,A -85,B 0,C 180,E1 -14349.577,E2 -14349.577} C_VEL
LIN {X 0,Y 333.63,Z 288.735,A -85,B 0,C 180,E1 -14352.499,E2 -14352.499} C_VEL
LIN {X 0,Y 333.668,Z 288.733,A -85,B 0,C 180,E1 -14355.967,E2 -14355.967} C_VEL
LIN {X 0,Y 333.697,Z 288.73,A -85,B 0,C 180,E1 -14359.303,E2 -14359.303} C_VEL
LIN {X 0,Y 333.66,Z 288.732,A -85,B 0,C 180,E1 -14363.167,E2 -14363.167} C_VEL
LIN {X 0,Y 333.63,Z 288.735,A -85,B 0,C 180,E1 -14366.791,E2 -14366.791} C_VEL
LIN {X 0,Y 333.696,Z 288.73,A -85,B 0,C 180,E1 -14369.709,E2 -14369.709} C_VEL
LIN {X 0,Y 333.737,Z 288.725,A -85,B 0,C 180,E1 -14372.4,E2 -14372.4} C_VEL
LIN {X 0,Y 333.718,Z 288.724,A -85,B 0,C 180,E1 -14375.09,E2 -14375.09} C_VEL
LIN {X 0,Y 333.67,Z 288.731,A -85,B 0,C 180,E1 -14379.018,E2 -14379.018} C_VEL
LIN {X 0,Y 333.785,Z 288.716,A -85,B 0,C 180,E1 -14381.589,E2 -14381.589} C_VEL
LIN {X 0,Y 333.799,Z 288.714,A -85,B 0,C 180,E1 -14385.576,E2 -14385.576} C_VEL
LIN {X 0,Y 333.823,Z 288.714,A -85,B 0,C 180,E1 -14389.078,E2 -14389.078} C_VEL
LIN {X 0,Y 333.996,Z 288.695,A -85,B 0,C 180,E1 -14392.747,E2 -14392.747} C_VEL
LIN {X 0,Y 333.798,Z 288.718,A -85,B 0,C 180,E1 -14395.169,E2 -14395.169} C_VEL
LIN {X 0,Y 334.096,Z 288.678,A -85,B 0,C 180,E1 -14397.589,E2 -14397.589} C_VEL
LIN {X 0,Y 334.236,Z 288.66,A -85,B 0,C 180,E1 -14400,E2 -14400} C_VEL
LIN {X 0,Y 334.094,Z 288.678,A -85,B 0,C 180,E1 -14402.411,E2 -14402.411} C_VEL
LIN {X 0,Y 334.004,Z 288.689,A -85,B 0,C 180,E1 -14406.039,E2 -14406.039} C_VEL
LIN {X 0,Y 333.85,Z 288.712,A -85,B 0,C 180,E1 -14409.695,E2 -14409.695} C_VEL
LIN {X 0,Y 333.789,Z 288.72,A -85,B 0,C 180,E1 -14413.392,E2 -14413.392} C_VEL
LIN {X 0,Y 333.736,Z 288.723,A -85,B 0,C 180,E1 -14417.147,E2 -14417.147} C_VEL
LIN {X 0,Y 333.722,Z 288.729,A -85,B 0,C 180,E1 -14419.691,E2 -14419.691} C_VEL
LIN {X 0,Y 333.662,Z 288.734,A -85,B 0,C 180,E1 -14423.591,E2 -14423.591} C_VEL
LIN {X 0,Y 333.726,Z 288.727,A -85,B 0,C 180,E1 -14426.247,E2 -14426.247} C_VEL
LIN {X 0,Y 333.682,Z 288.729,A -85,B 0,C 180,E1 -14428.975,E2 -14428.975} C_VEL
LIN {X 0,Y 333.635,Z 288.738,A -85,B 0,C 180,E1 -14432.587,E2 -14432.587} C_VEL
LIN {X 0,Y 333.668,Z 288.734,A -85,B 0,C 180,E1 -14436.14,E2 -14436.14} C_VEL
LIN {X 0,Y 333.64,Z 288.735,A -85,B 0,C 180,E1 -14439.193,E2 -14439.193} C_VEL
LIN {X 0,Y 333.627,Z 288.741,A -85,B 0,C 180,E1 -14442.501,E2 -14442.501} C_VEL
LIN {X 0,Y 333.613,Z 288.738,A -85,B 0,C 180,E1 -14445.96,E2 -14445.96} C_VEL
LIN {X 0,Y 333.642,Z 288.736,A -85,B 0,C 180,E1 -14449.316,E2 -14449.316} C_VEL
LIN {X 0,Y 333.66,Z 288.736,A -85,B 0,C 180,E1 -14453.169,E2 -14453.169} C_VEL
LIN {X 0,Y 333.67,Z 288.734,A -85,B 0,C 180,E1 -14455.342,E2 -14455.342} C_VEL
LIN {X 0,Y 333.626,Z 288.736,A -85,B 0,C 180,E1 -14458.222,E2 -14458.222} C_VEL
LIN {X 0,Y 333.652,Z 288.736,A -85,B 0,C 180,E1 -14461.023,E2 -14461.023} C_VEL
LIN {X 0,Y 333.727,Z 288.933,A -85,B 0,C 180,E1 -14463.079,E2 -14463.079} C_VEL
LIN {X 0,Y 335.791,Z 299.961,A -85,B 0,C 180,E1 -14466.568,E2 -14466.568} C_VEL
LIN {X 0,Y 335.651,Z 304.302,A -85,B 0,C 180,E1 -14467.859,E2 -14467.859} C_VEL
LIN {X 0,Y 334.391,Z 317.245,A -85,B 0,C 180,E1 -14471.624,E2 -14471.624} C_VEL
LIN {X 0,Y 338.539,Z 348.647,A -85,B 0,C 180,E1 -14472.54,E2 -14472.54} C_VEL
LIN {X 0,Y 337.821,Z 394.157,A -85,B 0,C 180,E1 -14473.562,E2 -14473.562} C_VEL
LIN {X 0,Y 337.356,Z 403.575,A -85,B 0,C 180,E1 -14473.913,E2 -14473.913} C_VEL
LIN {X 0,Y 336.753,Z 413.954,A -85,B 0,C 180,E1 -14474.491,E2 -14474.491} C_VEL
LIN {X 0,Y 336.079,Z 424.461,A -85,B 0,C 180,E1 -14475.312,E2 -14475.312} C_VEL
LIN {X 0,Y 335.229,Z 434.388,A -85,B 0,C 180,E1 -14476.358,E2 -14476.358} C_VEL
LIN {X 0,Y 334.524,Z 442.348,A -85,B 0,C 180,E1 -14477.411,E2 -14477.411} C_VEL
LIN {X 0,Y 333.927,Z 448.925,A -85,B 0,C 180,E1 -14478.467,E2 -14478.467} C_VEL
LIN {X 0,Y 333.287,Z 455.174,A -85,B 0,C 180,E1 -14479.675,E2 -14479.675} C_VEL
LIN {X 0,Y 332.817,Z 460.36,A -85,B 0,C 180,E1 -14480.888,E2 -14480.888} C_VEL
LIN {X 0,Y 332.474,Z 464.674,A -85,B 0,C 180,E1 -14482.103,E2 -14482.103} C_VEL
LIN {X 0,Y 332.22,Z 468.249,A -85,B 0,C 180,E1 -14483.319,E2 -14483.319} C_VEL
LIN {X 0,Y 332.047,Z 472.342,A -85,B 0,C 180,E1 -14485.144,E2 -14485.144} C_VEL
LIN {X 0,Y 332.021,Z 474.343,A -85,B 0,C 180,E1 -14486.359,E2 -14486.359} C_VEL
LIN {X 0,Y 331.922,Z 475.824,A -85,B 0,C 180,E1 -14487.573,E2 -14487.573} C_VEL
LIN {X 0,Y 331.912,Z 476.773,A -85,B 0,C 180,E1 -14488.787,E2 -14488.787} C_VEL
LIN {X 0,Y 331.967,Z 477.13,A -85,B 0,C 180,E1 -14490,E2 -14490} C_VEL
LIN {X 0,Y 331.91,Z 477.004,A -85,B 0,C 180,E1 -14491.213,E2 -14491.213} C_VEL
LIN {X 0,Y 331.92,Z 476.412,A -85,B 0,C 180,E1 -14492.427,E2 -14492.427} C_VEL
LIN {X 0,Y 332.021,Z 475.344,A -85,B 0,C 180,E1 -14493.641,E2 -14493.641} C_VEL
LIN {X 0,Y 332.061,Z 472.586,A -85,B 0,C 180,E1 -14495.481,E2 -14495.481} C_VEL
LIN {X 0,Y 332.422,Z 468.635,A -85,B 0,C 180,E1 -14497.287,E2 -14497.287} C_VEL
LIN {X 0,Y 332.717,Z 465.195,A -85,B 0,C 180,E1 -14498.503,E2 -14498.503} C_VEL
LIN {X 0,Y 333.301,Z 459.857,A -85,B 0,C 180,E1 -14500.018,E2 -14500.018} C_VEL
LIN {X 0,Y 333.89,Z 454.627,A -85,B 0,C 180,E1 -14501.227,E2 -14501.227} C_VEL
LIN {X 0,Y 334.662,Z 448.348,A -85,B 0,C 180,E1 -14502.43,E2 -14502.43} C_VEL
LIN {X 0,Y 335.489,Z 440.725,A -85,B 0,C 180,E1 -14503.631,E2 -14503.631} C_VEL
LIN {X 0,Y 336.565,Z 431.267,A -85,B 0,C 180,E1 -14504.82,E2 -14504.82} C_VEL
LIN {X 0,Y 337.443,Z 422.075,A -85,B 0,C 180,E1 -14505.709,E2 -14505.709} C_VEL
LIN {X 0,Y 338.15,Z 412.062,A -85,B 0,C 180,E1 -14506.449,E2 -14506.449} C_VEL
LIN {X 0,Y 338.843,Z 402.353,A -85,B 0,C 180,E1 -14506.967,E2 -14506.967} C_VEL
LIN {X 0,Y 339.307,Z 393.424,A -85,B 0,C 180,E1 -14507.29,E2 -14507.29} C_VEL
LIN {X 0,Y 339.965,Z 347.366,A -85,B 0,C 180,E1 -14508.341,E2 -14508.341} C_VEL
LIN {X 0,Y 336.379,Z 323.818,A -85,B 0,C 180,E1 -14509.121,E2 -14509.121} C_VEL
LIN {X 0,Y 335.007,Z 316.36,A -85,B 0,C 180,E1 -14509.392,E2 -14509.392} C_VEL
LIN {X 0,Y 336.222,Z 303.273,A -85,B 0,C 180,E1 -14513.114,E2 -14513.114} C_VEL
LIN {X 0,Y 335.547,Z 297.867,A -85,B 0,C 180,E1 -14514.764,E2 -14514.764} C_VEL
LIN {X 0,Y 333.638,Z 288.74,A -85,B 0,C 180,E1 -14517.703,E2 -14517.703} C_VEL
LIN {X 0,Y 333.653,Z 288.741,A -85,B 0,C 180,E1 -14520.365,E2 -14520.365} C_VEL
LIN {X 0,Y 333.633,Z 288.739,A -85,B 0,C 180,E1 -14523.208,E2 -14523.208} C_VEL
LIN {X 0,Y 333.671,Z 288.735,A -85,B 0,C 180,E1 -14526.138,E2 -14526.138} C_VEL
LIN {X 0,Y 333.641,Z 288.742,A -85,B 0,C 180,E1 -14529.192,E2 -14529.192} C_VEL
LIN {X 0,Y 333.626,Z 288.74,A -85,B 0,C 180,E1 -14532.499,E2 -14532.499} C_VEL
LIN {X 0,Y 333.59,Z 288.745,A -85,B 0,C 180,E1 -14535.954,E2 -14535.954} C_VEL
LIN {X 0,Y 333.64,Z 288.734,A -85,B 0,C 180,E1 -14539.315,E2 -14539.315} C_VEL
LIN {X 0,Y 333.657,Z 288.728,A -85,B 0,C 180,E1 -14543.167,E2 -14543.167} C_VEL
LIN {X 0,Y 333.666,Z 288.735,A -85,B 0,C 180,E1 -14545.341,E2 -14545.341} C_VEL
LIN {X 0,Y 333.695,Z 288.731,A -85,B 0,C 180,E1 -14549.71,E2 -14549.71} C_VEL
LIN {X 0,Y 333.733,Z 288.714,A -85,B 0,C 180,E1 -14552.4,E2 -14552.4} C_VEL
LIN {X 0,Y 333.716,Z 288.725,A -85,B 0,C 180,E1 -14555.09,E2 -14555.09} C_VEL
LIN {X 0,Y 333.663,Z 288.726,A -85,B 0,C 180,E1 -14559.018,E2 -14559.018} C_VEL
LIN {X 0,Y 333.784,Z 288.718,A -85,B 0,C 180,E1 -14561.589,E2 -14561.589} C_VEL
LIN {X 0,Y 333.799,Z 288.709,A -85,B 0,C 180,E1 -14565.576,E2 -14565.576} C_VEL
LIN {X 0,Y 333.823,Z 288.707,A -85,B 0,C 180,E1 -14569.078,E2 -14569.078} C_VEL
LIN {X 0,Y 333.996,Z 288.69,A -85,B 0,C 180,E1 -14572.747,E2 -14572.747} C_VEL
LIN {X 0,Y 333.796,Z 288.71,A -85,B 0,C 180,E1 -14575.169,E2 -14575.169} C_VEL
LIN {X 0,Y 334.093,Z 288.673,A -85,B 0,C 180,E1 -14577.589,E2 -14577.589} C_VEL
LIN {X 0,Y 334.235,Z 288.659,A -85,B 0,C 180,E1 -14580,E2 -14580} C_VEL
LIN {X 0,Y 334.093,Z 288.668,A -85,B 0,C 180,E1 -14582.411,E2 -14582.411} C_VEL
LIN {X 0,Y 333.958,Z 288.69,A -85,B 0,C 180,E1 -14586.495,E2 -14586.495} C_VEL
LIN {X 0,Y 333.839,Z 288.713,A -85,B 0,C 180,E1 -14589.696,E2 -14589.696} C_VEL
LIN {X 0,Y 333.787,Z 288.715,A -85,B 0,C 180,E1 -14593.392,E2 -14593.392} C_VEL
LIN {X 0,Y 333.736,Z 288.72,A -85,B 0,C 180,E1 -14597.147,E2 -14597.147} C_VEL
LIN {X 0,Y 333.726,Z 288.727,A -85,B 0,C 180,E1 -14599.691,E2 -14599.691} C_VEL
LIN {X 0,Y 333.684,Z 288.735,A -85,B 0,C 180,E1 -14602.279,E2 -14602.279} C_VEL
LIN {X 0,Y 333.728,Z 288.726,A -85,B 0,C 180,E1 -14606.247,E2 -14606.247} C_VEL
LIN {X 0,Y 333.704,Z 288.726,A -85,B 0,C 180,E1 -14608.973,E2 -14608.973} C_VEL
LIN {X 0,Y 333.636,Z 288.739,A -85,B 0,C 180,E1 -14612.588,E2 -14612.588} C_VEL
LIN {X 0,Y 333.67,Z 288.735,A -85,B 0,C 180,E1 -14616.14,E2 -14616.14} C_VEL
LIN {X 0,Y 333.709,Z 288.889,A -85,B 0,C 180,E1 -14619.281,E2 -14619.281} C_VEL
LIN {X 0,Y 335.479,Z 297.599,A -85,B 0,C 180,E1 -14622.096,E2 -14622.096} C_VEL
LIN {X 0,Y 335.59,Z 299.525,A -85,B 0,C 180,E1 -14622.686,E2 -14622.686} C_VEL
LIN {X 0,Y 340.15,Z 321.505,A -85,B 0,C 180,E1 -14623.514,E2 -14623.514} C_VEL
LIN {X 0,Y 340.5,Z 326.039,A -85,B 0,C 180,E1 -14623.642,E2 -14623.642} C_VEL
LIN {X 0,Y 339.428,Z 376.25,A -85,B 0,C 180,E1 -14624.769,E2 -14624.769} C_VEL
LIN {X 0,Y 339.009,Z 386.341,A -85,B 0,C 180,E1 -14625.156,E2 -14625.156} C_VEL
LIN {X 0,Y 338.451,Z 397.675,A -85,B 0,C 180,E1 -14625.82,E2 -14625.82} C_VEL
LIN {X 0,Y 337.686,Z 407.406,A -85,B 0,C 180,E1 -14626.624,E2 -14626.624} C_VEL
LIN {X 0,Y 336.891,Z 415.865,A -85,B 0,C 180,E1 -14627.518,E2 -14627.518} C_VEL
LIN {X 0,Y 336.038,Z 423.597,A -85,B 0,C 180,E1 -14628.526,E2 -14628.526} C_VEL
LIN {X 0,Y 335.209,Z 430.708,A -85,B 0,C 180,E1 -14629.661,E2 -14629.661} C_VEL
LIN {X 0,Y 334.428,Z 437.154,A -85,B 0,C 180,E1 -14630.918,E2 -14630.918} C_VEL
LIN {X 0,Y 333.71,Z 443.15,A -85,B 0,C 180,E1 -14632.358,E2 -14632.358} C_VEL
LIN {X 0,Y 333.181,Z 447.954,A -85,B 0,C 180,E1 -14633.8,E2 -14633.8} C_VEL
LIN {X 0,Y 332.583,Z 452.385,A -85,B 0,C 180,E1 -14635.501,E2 -14635.501} C_VEL
LIN {X 0,Y 332.41,Z 454.595,A -85,B 0,C 180,E1 -14636.654,E2 -14636.654} C_VEL
LIN {X 0,Y 332.142,Z 456.67,A -85,B 0,C 180,E1 -14638.064,E2 -14638.064} C_VEL
LIN {X 0,Y 331.823,Z 458.561,A -85,B 0,C 180,E1 -14640.271,E2 -14640.271} C_VEL
LIN {X 0,Y 331.737,Z 458.571,A -85,B 0,C 180,E1 -14642.847,E2 -14642.847} C_VEL
LIN {X 0,Y 331.899,Z 456.95,A -85,B 0,C 180,E1 -14644.945,E2 -14644.945} C_VEL
LIN {X 0,Y 332.095,Z 455.092,A -85,B 0,C 180,E1 -14646.292,E2 -14646.292} C_VEL
LIN {X 0,Y 332.357,Z 452.539,A -85,B 0,C 180,E1 -14647.628,E2 -14647.628} C_VEL
LIN {X 0,Y 332.811,Z 447.314,A -85,B 0,C 180,E1 -14649.609,E2 -14649.609} C_VEL
LIN {X 0,Y 333.205,Z 442.865,A -85,B 0,C 180,E1 -14650.919,E2 -14650.919} C_VEL
LIN {X 0,Y 333.729,Z 437.443,A -85,B 0,C 180,E1 -14652.221,E2 -14652.221} C_VEL
LIN {X 0,Y 334.363,Z 430.836,A -85,B 0,C 180,E1 -14653.516,E2 -14653.516} C_VEL
LIN {X 0,Y 334.927,Z 424.708,A -85,B 0,C 180,E1 -14654.514,E2 -14654.514} C_VEL
LIN {X 0,Y 335.683,Z 416.567,A -85,B 0,C 180,E1 -14655.605,E2 -14655.605} C_VEL
LIN {X 0,Y 336.406,Z 407.672,A -85,B 0,C 180,E1 -14656.561,E2 -14656.561} C_VEL
LIN {X 0,Y 337.115,Z 396.067,A -85,B 0,C 180,E1 -14657.509,E2 -14657.509} C_VEL
LIN {X 0,Y 337.591,Z 385.6,A -85,B 0,C 180,E1 -14658.103,E2 -14658.103} C_VEL
LIN {X 0,Y 337.963,Z 376.038,A -85,B 0,C 180,E1 -14658.468,E2 -14658.468} C_VEL
LIN {X 0,Y 338.67,Z 322.061,A -85,B 0,C 180,E1 -14659.682,E2 -14659.682} C_VEL
LIN {X 0,Y 334.705,Z 299.716,A -85,B 0,C 180,E1 -14660.399,E2 -14660.399} C_VEL
LIN {X 0,Y 334.82,Z 294.34,A -85,B 0,C 180,E1 -14662.159,E2 -14662.159} C_VEL
LIN {X 0,Y 334.014,Z 288.693,A -85,B 0,C 180,E1 -14664.113,E2 -14664.113} C_VEL
LIN {X 0,Y 334.107,Z 288.68,A -85,B 0,C 180,E1 -14667.589,E2 -14667.589} C_VEL
LIN {X 0,Y 334.248,Z 288.664,A -85,B 0,C 180,E1 -14670,E2 -14670} C_VEL
LIN {X 0,Y 334.107,Z 288.678,A -85,B 0,C 180,E1 -14672.411,E2 -14672.411} C_VEL
LIN {X 0,Y 334.003,Z 288.694,A -85,B 0,C 180,E1 -14676.039,E2 -14676.039} C_VEL
LIN {X 0,Y 333.851,Z 288.709,A -85,B 0,C 180,E1 -14679.695,E2 -14679.695} C_VEL
LIN {X 0,Y 333.798,Z 288.714,A -85,B 0,C 180,E1 -14683.391,E2 -14683.391} C_VEL
LIN {X 0,Y 333.719,Z 288.725,A -85,B 0,C 180,E1 -14687.147,E2 -14687.147} C_VEL
LIN {X 0,Y 333.685,Z 288.728,A -85,B 0,C 180,E1 -14689.693,E2 -14689.693} C_VEL
LIN {X 0,Y 333.669,Z 288.73,A -85,B 0,C 180,E1 -14693.589,E2 -14693.589} C_VEL
LIN {X 0,Y 333.734,Z 288.723,A -85,B 0,C 180,E1 -14696.246,E2 -14696.246} C_VEL
LIN {X 0,Y 333.709,Z 288.732,A -85,B 0,C 180,E1 -14698.971,E2 -14698.971} C_VEL
LIN {X 0,Y 333.641,Z 288.736,A -85,B 0,C 180,E1 -14702.586,E2 -14702.586} C_VEL
LIN {X 0,Y 333.673,Z 288.73,A -85,B 0,C 180,E1 -14706.138,E2 -14706.138} C_VEL
LIN {X 0,Y 333.622,Z 288.738,A -85,B 0,C 180,E1 -14709.577,E2 -14709.577} C_VEL
LIN {X 0,Y 332.934,Z 288.823,A -85,B 0,C 180,E1 -14710.585,E2 -14710.585} C_VEL
LIN {X 0,Y 330.074,Z 289.178,A -85,B 0,C 180,E1 -14712.226,E2 -14712.226} C_VEL
LIN {X 0,Y 327.672,Z 289.483,A -85,B 0,C 180,E1 -14713.554,E2 -14713.554} C_VEL
LIN {X 0,Y 326.657,Z 289.604,A -85,B 0,C 180,E1 -14714.583,E2 -14714.583} C_VEL
LIN {X 0,Y 326.582,Z 289.614,A -85,B 0,C 180,E1 -14714.931,E2 -14714.931} C_VEL
LIN {X 0,Y 326.618,Z 289.61,A -85,B 0,C 180,E1 -14718.161,E2 -14718.161} C_VEL
LIN {X 0,Y 326.639,Z 289.609,A -85,B 0,C 180,E1 -14721.393,E2 -14721.393} C_VEL
LIN {X 0,Y 326.613,Z 289.609,A -85,B 0,C 180,E1 -14724.85,E2 -14724.85} C_VEL
LIN {X 0,Y 326.601,Z 289.612,A -85,B 0,C 180,E1 -14727.455,E2 -14727.455} C_VEL
LIN {X 0,Y 326.654,Z 289.608,A -85,B 0,C 180,E1 -14730.34,E2 -14730.34} C_VEL
LIN {X 0,Y 326.682,Z 289.604,A -85,B 0,C 180,E1 -14734.515,E2 -14734.515} C_VEL
LIN {X 0,Y 326.637,Z 289.61,A -85,B 0,C 180,E1 -14738.544,E2 -14738.544} C_VEL
LIN {X 0,Y 326.736,Z 289.594,A -85,B 0,C 180,E1 -14741.177,E2 -14741.177} C_VEL
LIN {X 0,Y 326.754,Z 289.592,A -85,B 0,C 180,E1 -14745.433,E2 -14745.433} C_VEL
LIN {X 0,Y 326.76,Z 289.596,A -85,B 0,C 180,E1 -14748.838,E2 -14748.838} C_VEL
LIN {X 0,Y 326.949,Z 289.571,A -85,B 0,C 180,E1 -14752.59,E2 -14752.59} C_VEL
LIN {X 0,Y 326.765,Z 289.595,A -85,B 0,C 180,E1 -14755.065,E2 -14755.065} C_VEL
LIN {X 0,Y 327.036,Z 289.558,A -85,B 0,C 180,E1 -14757.537,E2 -14757.537} C_VEL
LIN {X 0,Y 327.187,Z 289.538,A -85,B 0,C 180,E1 -14760,E2 -14760} C_VEL
LIN {X 0,Y 327.035,Z 289.557,A -85,B 0,C 180,E1 -14762.463,E2 -14762.463} C_VEL
LIN {X 0,Y 326.978,Z 289.564,A -85,B 0,C 180,E1 -14766.169,E2 -14766.169} C_VEL
LIN {X 0,Y 326.803,Z 289.587,A -85,B 0,C 180,E1 -14769.906,E2 -14769.906} C_VEL
LIN {X 0,Y 326.751,Z 289.598,A -85,B 0,C 180,E1 -14773.686,E2 -14773.686} C_VEL
LIN {X 0,Y 326.69,Z 289.604,A -85,B 0,C 180,E1 -14777.528,E2 -14777.528} C_VEL
LIN {X 0,Y 326.648,Z 289.608,A -85,B 0,C 180,E1 -14780.136,E2 -14780.136} C_VEL
LIN {X 0,Y 326.641,Z 289.61,A -85,B 0,C 180,E1 -14784.13,E2 -14784.13} C_VEL
LIN {X 0,Y 326.674,Z 289.602,A -85,B 0,C 180,E1 -14786.858,E2 -14786.858} C_VEL
LIN {X 0,Y 326.626,Z 289.61,A -85,B 0,C 180,E1 -14790.61,E2 -14790.61} C_VEL
LIN {X 0,Y 326.599,Z 289.614,A -85,B 0,C 180,E1 -14794.02,E2 -14794.02} C_VEL
LIN {X 0,Y 326.62,Z 289.609,A -85,B 0,C 180,E1 -14797.239,E2 -14797.239} C_VEL
LIN {X 0,Y 326.571,Z 289.615,A -85,B 0,C 180,E1 -14801.132,E2 -14801.132} C_VEL
LIN {X 0,Y 326.551,Z 289.623,A -85,B 0,C 180,E1 -14804.749,E2 -14804.749} C_VEL
LIN {X 0,Y 326.571,Z 289.615,A -85,B 0,C 180,E1 -14808.155,E2 -14808.155} C_VEL
LIN {X 0,Y 326.593,Z 289.614,A -85,B 0,C 180,E1 -14811.389,E2 -14811.389} C_VEL
LIN {X 0,Y 326.615,Z 289.613,A -85,B 0,C 180,E1 -14814.852,E2 -14814.852} C_VEL
LIN {X 0,Y 326.604,Z 289.614,A -85,B 0,C 180,E1 -14817.456,E2 -14817.456} C_VEL
LIN {X 0,Y 326.614,Z 289.609,A -85,B 0,C 180,E1 -14820.337,E2 -14820.337} C_VEL
LIN {X 0,Y 326.654,Z 289.658,A -85,B 0,C 180,E1 -14822.795,E2 -14822.795} C_VEL
LIN {X 0,Y 328.775,Z 301.04,A -85,B 0,C 180,E1 -14826.481,E2 -14826.481} C_VEL
LIN {X 0,Y 328.537,Z 306.107,A -85,B 0,C 180,E1 -14828.016,E2 -14828.016} C_VEL
LIN {X 0,Y 327.439,Z 317.064,A -85,B 0,C 180,E1 -14831.27,E2 -14831.27} C_VEL
LIN {X 0,Y 331.694,Z 348.819,A -85,B 0,C 180,E1 -14832.22,E2 -14832.22} C_VEL
LIN {X 0,Y 330.972,Z 393.892,A -85,B 0,C 180,E1 -14833.254,E2 -14833.254} C_VEL
LIN {X 0,Y 330.525,Z 402.889,A -85,B 0,C 180,E1 -14833.593,E2 -14833.593} C_VEL
LIN {X 0,Y 329.996,Z 411.867,A -85,B 0,C 180,E1 -14834.086,E2 -14834.086} C_VEL
LIN {X 0,Y 329.328,Z 422.03,A -85,B 0,C 180,E1 -14834.846,E2 -14834.846} C_VEL
LIN {X 0,Y 328.407,Z 432.604,A -85,B 0,C 180,E1 -14835.911,E2 -14835.911} C_VEL
LIN {X 0,Y 327.653,Z 440.832,A -85,B 0,C 180,E1 -14836.985,E2 -14836.985} C_VEL
LIN {X 0,Y 326.933,Z 448.486,A -85,B 0,C 180,E1 -14838.217,E2 -14838.217} C_VEL
LIN {X 0,Y 326.299,Z 454.778,A -85,B 0,C 180,E1 -14839.451,E2 -14839.451} C_VEL
LIN {X 0,Y 325.799,Z 459.999,A -85,B 0,C 180,E1 -14840.69,E2 -14840.69} C_VEL
LIN {X 0,Y 325.433,Z 464.345,A -85,B 0,C 180,E1 -14841.931,E2 -14841.931} C_VEL
LIN {X 0,Y 325.055,Z 469.479,A -85,B 0,C 180,E1 -14843.794,E2 -14843.794} C_VEL
LIN {X 0,Y 324.942,Z 473.219,A -85,B 0,C 180,E1 -14845.659,E2 -14845.659} C_VEL
LIN {X 0,Y 324.843,Z 475.595,A -85,B 0,C 180,E1 -14847.52,E2 -14847.52} C_VEL
LIN {X 0,Y 324.821,Z 476.549,A -85,B 0,C 180,E1 -14848.76,E2 -14848.76} C_VEL
LIN {X 0,Y 324.872,Z 476.922,A -85,B 0,C 180,E1 -14850,E2 -14850} C_VEL
LIN {X 0,Y 324.82,Z 476.817,A -85,B 0,C 180,E1 -14851.24,E2 -14851.24} C_VEL
LIN {X 0,Y 324.841,Z 476.246,A -85,B 0,C 180,E1 -14852.48,E2 -14852.48} C_VEL
LIN {X 0,Y 324.928,Z 475.195,A -85,B 0,C 180,E1 -14853.72,E2 -14853.72} C_VEL
LIN {X 0,Y 324.96,Z 473.547,A -85,B 0,C 180,E1 -14854.963,E2 -14854.963} C_VEL
LIN {X 0,Y 325.201,Z 470.077,A -85,B 0,C 180,E1 -14856.826,E2 -14856.826} C_VEL
LIN {X 0,Y 325.681,Z 465.135,A -85,B 0,C 180,E1 -14858.688,E2 -14858.688} C_VEL
LIN {X 0,Y 326.287,Z 459.835,A -85,B 0,C 180,E1 -14860.235,E2 -14860.235} C_VEL
LIN {X 0,Y 326.926,Z 454.645,A -85,B 0,C 180,E1 -14861.469,E2 -14861.469} C_VEL
LIN {X 0,Y 327.73,Z 448.408,A -85,B 0,C 180,E1 -14862.697,E2 -14862.697} C_VEL
LIN {X 0,Y 328.489,Z 441.859,A -85,B 0,C 180,E1 -14863.769,E2 -14863.769} C_VEL
LIN {X 0,Y 329.42,Z 433.94,A -85,B 0,C 180,E1 -14864.833,E2 -14864.833} C_VEL
LIN {X 0,Y 330.505,Z 424.083,A -85,B 0,C 180,E1 -14865.889,E2 -14865.889} C_VEL
LIN {X 0,Y 331.372,Z 412.586,A -85,B 0,C 180,E1 -14866.796,E2 -14866.796} C_VEL
LIN {X 0,Y 332.119,Z 402.622,A -85,B 0,C 180,E1 -14867.346,E2 -14867.346} C_VEL
LIN {X 0,Y 332.639,Z 392.906,A -85,B 0,C 180,E1 -14867.706,E2 -14867.706} C_VEL
LIN {X 0,Y 333.298,Z 347.932,A -85,B 0,C 180,E1 -14868.755,E2 -14868.755} C_VEL
LIN {X 0,Y 329.811,Z 325.002,A -85,B 0,C 180,E1 -14869.538,E2 -14869.538} C_VEL
LIN {X 0,Y 328.135,Z 316.037,A -85,B 0,C 180,E1 -14869.906,E2 -14869.906} C_VEL
LIN {X 0,Y 329.308,Z 303.987,A -85,B 0,C 180,E1 -14873.409,E2 -14873.409} C_VEL
LIN {X 0,Y 328.291,Z 297.855,A -85,B 0,C 180,E1 -14875.35,E2 -14875.35} C_VEL
LIN {X 0,Y 326.622,Z 289.616,A -85,B 0,C 180,E1 -14878.091,E2 -14878.091} C_VEL
LIN {X 0,Y 326.569,Z 289.617,A -85,B 0,C 180,E1 -14881.096,E2 -14881.096} C_VEL
LIN {X 0,Y 326.603,Z 289.614,A -85,B 0,C 180,E1 -14884.019,E2 -14884.019} C_VEL
LIN {X 0,Y 326.623,Z 289.615,A -85,B 0,C 180,E1 -14887.238,E2 -14887.238} C_VEL
LIN {X 0,Y 326.572,Z 289.625,A -85,B 0,C 180,E1 -14891.13,E2 -14891.13} C_VEL
LIN {X 0,Y 326.521,Z 289.628,A -85,B 0,C 180,E1 -14894.742,E2 -14894.742} C_VEL
LIN {X 0,Y 326.569,Z 289.615,A -85,B 0,C 180,E1 -14898.153,E2 -14898.153} C_VEL
LIN {X 0,Y 326.616,Z 289.613,A -85,B 0,C 180,E1 -14901.391,E2 -14901.391} C_VEL
LIN {X 0,Y 326.611,Z 289.611,A -85,B 0,C 180,E1 -14904.851,E2 -14904.851} C_VEL
LIN {X 0,Y 326.6,Z 289.606,A -85,B 0,C 180,E1 -14907.455,E2 -14907.455} C_VEL
LIN {X 0,Y 326.652,Z 289.606,A -85,B 0,C 180,E1 -14910.34,E2 -14910.34} C_VEL
LIN {X 0,Y 326.681,Z 289.603,A -85,B 0,C 180,E1 -14914.516,E2 -14914.516} C_VEL
LIN {X 0,Y 326.61,Z 289.602,A -85,B 0,C 180,E1 -14918.543,E2 -14918.543} C_VEL
LIN {X 0,Y 326.736,Z 289.595,A -85,B 0,C 180,E1 -14921.177,E2 -14921.177} C_VEL
LIN {X 0,Y 326.754,Z 289.586,A -85,B 0,C 180,E1 -14925.433,E2 -14925.433} C_VEL
LIN {X 0,Y 326.759,Z 289.589,A -85,B 0,C 180,E1 -14928.839,E2 -14928.839} C_VEL
LIN {X 0,Y 326.948,Z 289.566,A -85,B 0,C 180,E1 -14932.59,E2 -14932.59} C_VEL
LIN {X 0,Y 326.763,Z 289.587,A -85,B 0,C 180,E1 -14935.065,E2 -14935.065} C_VEL
LIN {X 0,Y 327.034,Z 289.552,A -85,B 0,C 180,E1 -14937.537,E2 -14937.537} C_VEL
LIN {X 0,Y 327.187,Z 289.537,A -85,B 0,C 180,E1 -14940,E2 -14940} C_VEL
LIN {X 0,Y 327.034,Z 289.547,A -85,B 0,C 180,E1 -14942.463,E2 -14942.463} C_VEL
LIN {X 0,Y 326.919,Z 289.567,A -85,B 0,C 180,E1 -14946.484,E2 -14946.484} C_VEL
LIN {X 0,Y 326.794,Z 289.59,A -85,B 0,C 180,E1 -14949.907,E2 -14949.907} C_VEL
LIN {X 0,Y 326.749,Z 289.595,A -85,B 0,C 180,E1 -14953.686,E2 -14953.686} C_VEL
LIN {X 0,Y 326.689,Z 289.601,A -85,B 0,C 180,E1 -14957.529,E2 -14957.529} C_VEL
LIN {X 0,Y 326.653,Z 289.605,A -85,B 0,C 180,E1 -14960.136,E2 -14960.136} C_VEL
LIN {X 0,Y 326.643,Z 289.61,A -85,B 0,C 180,E1 -14964.13,E2 -14964.13} C_VEL
LIN {X 0,Y 326.677,Z 289.602,A -85,B 0,C 180,E1 -14966.858,E2 -14966.858} C_VEL
LIN {X 0,Y 326.632,Z 289.609,A -85,B 0,C 180,E1 -14970.612,E2 -14970.612} C_VEL
LIN {X 0,Y 326.6,Z 289.616,A -85,B 0,C 180,E1 -14974.02,E2 -14974.02} C_VEL
LIN {X 0,Y 326.623,Z 289.613,A -85,B 0,C 180,E1 -14977.24,E2 -14977.24} C_VEL
LIN {X 0,Y 326.668,Z 289.641,A -85,B 0,C 180,E1 -14978.868,E2 -14978.868} C_VEL
LIN {X 0,Y 328.625,Z 299.557,A -85,B 0,C 180,E1 -14982.144,E2 -14982.144} C_VEL
LIN {X 0,Y 328.747,Z 300.243,A -85,B 0,C 180,E1 -14982.228,E2 -14982.228} C_VEL
LIN {X 0,Y 332.469,Z 316.857,A -85,B 0,C 180,E1 -14982.895,E2 -14982.895} C_VEL
LIN {X 0,Y 333.885,Z 325.088,A -85,B 0,C 180,E1 -14983.187,E2 -14983.187} C_VEL
LIN {X 0,Y 332.754,Z 376.798,A -85,B 0,C 180,E1 -14984.375,E2 -14984.375} C_VEL
LIN {X 0,Y 332.284,Z 386.979,A -85,B 0,C 180,E1 -14984.778,E2 -14984.778} C_VEL
LIN {X 0,Y 331.641,Z 399.014,A -85,B 0,C 180,E1 -14985.523,E2 -14985.523} C_VEL
LIN {X 0,Y 330.853,Z 408.406,A -85,B 0,C 180,E1 -14986.335,E2 -14986.335} C_VEL
LIN {X 0,Y 330.025,Z 416.733,A -85,B 0,C 180,E1 -14987.247,E2 -14987.247} C_VEL
LIN {X 0,Y 329.264,Z 423.397,A -85,B 0,C 180,E1 -14988.133,E2 -14988.133} C_VEL
LIN {X 0,Y 328.411,Z 430.385,A -85,B 0,C 180,E1 -14989.256,E2 -14989.256} C_VEL
LIN {X 0,Y 327.543,Z 437.087,A -85,B 0,C 180,E1 -14990.574,E2 -14990.574} C_VEL
LIN {X 0,Y 326.719,Z 443.636,A -85,B 0,C 180,E1 -14992.177,E2 -14992.177} C_VEL
LIN {X 0,Y 326.156,Z 448.425,A -85,B 0,C 180,E1 -14993.662,E2 -14993.662} C_VEL
LIN {X 0,Y 325.594,Z 452.108,A -85,B 0,C 180,E1 -14995.109,E2 -14995.109} C_VEL
LIN {X 0,Y 325.358,Z 454.953,A -85,B 0,C 180,E1 -14996.578,E2 -14996.578} C_VEL
LIN {X 0,Y 324.934,Z 457.74,A -85,B 0,C 180,E1 -14998.729,E2 -14998.729} C_VEL
LIN {X 0,Y 324.745,Z 458.748,A -85,B 0,C 180,E1 -15000.149,E2 -15000.149} C_VEL
LIN {X 0,Y 324.649,Z 459.078,A -85,B 0,C 180,E1 -15001.56,E2 -15001.56} C_VEL
LIN {X 0,Y 324.644,Z 458.73,A -85,B 0,C 180,E1 -15002.961,E2 -15002.961} C_VEL
LIN {X 0,Y 324.73,Z 457.743,A -85,B 0,C 180,E1 -15004.352,E2 -15004.352} C_VEL
LIN {X 0,Y 325.047,Z 455.149,A -85,B 0,C 180,E1 -15006.423,E2 -15006.423} C_VEL
LIN {X 0,Y 325.388,Z 451.483,A -85,B 0,C 180,E1 -15008.241,E2 -15008.241} C_VEL
LIN {X 0,Y 325.758,Z 447.271,A -85,B 0,C 180,E1 -15009.807,E2 -15009.807} C_VEL
LIN {X 0,Y 326.294,Z 441.828,A -85,B 0,C 180,E1 -15011.39,E2 -15011.39} C_VEL
LIN {X 0,Y 326.894,Z 435.745,A -85,B 0,C 180,E1 -15012.806,E2 -15012.806} C_VEL
LIN {X 0,Y 327.686,Z 427.763,A -85,B 0,C 180,E1 -15014.302,E2 -15014.302} C_VEL
LIN {X 0,Y 328.572,Z 418.758,A -85,B 0,C 180,E1 -15015.603,E2 -15015.603} C_VEL
LIN {X 0,Y 329.315,Z 410.283,A -85,B 0,C 180,E1 -15016.581,E2 -15016.581} C_VEL
LIN {X 0,Y 329.934,Z 401.488,A -85,B 0,C 180,E1 -15017.389,E2 -15017.389} C_VEL
LIN {X 0,Y 330.336,Z 393.714,A -85,B 0,C 180,E1 -15017.955,E2 -15017.955} C_VEL
LIN {X 0,Y 330.803,Z 384.085,A -85,B 0,C 180,E1 -15018.477,E2 -15018.477} C_VEL
LIN {X 0,Y 331.134,Z 374.227,A -85,B 0,C 180,E1 -15018.832,E2 -15018.832} C_VEL
LIN {X 0,Y 331.868,Z 322.988,A -85,B 0,C 180,E1 -15019.994,E2 -15019.994} C_VEL
LIN {X 0,Y 327.772,Z 299.907,A -85,B 0,C 180,E1 -15020.753,E2 -15020.753} C_VEL
LIN {X 0,Y 327.892,Z 296.196,A -85,B 0,C 180,E1 -15021.992,E2 -15021.992} C_VEL
LIN {X 0,Y 326.909,Z 289.578,A -85,B 0,C 180,E1 -15024.371,E2 -15024.371} C_VEL
LIN {X 0,Y 327.047,Z 289.559,A -85,B 0,C 180,E1 -15027.537,E2 -15027.537} C_VEL
LIN {X 0,Y 327.199,Z 289.542,A -85,B 0,C 180,E1 -15030,E2 -15030} C_VEL
LIN {X 0,Y 327.048,Z 289.557,A -85,B 0,C 180,E1 -15032.463,E2 -15032.463} C_VEL
LIN {X 0,Y 326.956,Z 289.573,A -85,B 0,C 180,E1 -15036.17,E2 -15036.17} C_VEL
LIN {X 0,Y 326.806,Z 289.588,A -85,B 0,C 180,E1 -15039.906,E2 -15039.906} C_VEL
LIN {X 0,Y 326.76,Z 289.591,A -85,B 0,C 180,E1 -15043.685,E2 -15043.685} C_VEL
LIN {X 0,Y 326.664,Z 289.603,A -85,B 0,C 180,E1 -15047.529,E2 -15047.529} C_VEL
LIN {X 0,Y 326.631,Z 289.609,A -85,B 0,C 180,E1 -15050.136,E2 -15050.136} C_VEL
LIN {X 0,Y 326.649,Z 289.606,A -85,B 0,C 180,E1 -15054.128,E2 -15054.128} C_VEL
LIN {X 0,Y 326.683,Z 289.607,A -85,B 0,C 180,E1 -15056.857,E2 -15056.857} C_VEL
LIN {X 0,Y 326.637,Z 289.609,A -85,B 0,C 180,E1 -15060.61,E2 -15060.61} C_VEL
LIN {X 0,Y 326.605,Z 289.61,A -85,B 0,C 180,E1 -15064.018,E2 -15064.018} C_VEL
LIN {X 0,Y 326.624,Z 289.615,A -85,B 0,C 180,E1 -15067.237,E2 -15067.237} C_VEL
LIN {X 0,Y 326.575,Z 289.618,A -85,B 0,C 180,E1 -15071.13,E2 -15071.13} C_VEL
LIN {X 0,Y 326.582,Z 289.614,A -85,B 0,C 180,E1 -15074.931,E2 -15074.931} C_VEL
LIN {X 0,Y 325.95,Z 289.699,A -85,B 0,C 180,E1 -15075.961,E2 -15075.961} C_VEL
LIN {X 0,Y 323.155,Z 290.051,A -85,B 0,C 180,E1 -15077.639,E2 -15077.639} C_VEL
LIN {X 0,Y 320.749,Z 290.348,A -85,B 0,C 180,E1 -15078.998,E2 -15078.998} C_VEL
LIN {X 0,Y 319.681,Z 290.476,A -85,B 0,C 180,E1 -15080.049,E2 -15080.049} C_VEL
LIN {X 0,Y 319.576,Z 290.486,A -85,B 0,C 180,E1 -15080.406,E2 -15080.406} C_VEL
LIN {X 0,Y 319.553,Z 290.492,A -85,B 0,C 180,E1 -15083.571,E2 -15083.571} C_VEL
LIN {X 0,Y 319.571,Z 290.486,A -85,B 0,C 180,E1 -15086.686,E2 -15086.686} C_VEL
LIN {X 0,Y 319.585,Z 290.487,A -85,B 0,C 180,E1 -15089.616,E2 -15089.616} C_VEL
LIN {X 0,Y 319.602,Z 290.485,A -85,B 0,C 180,E1 -15092.497,E2 -15092.497} C_VEL
LIN {X 0,Y 319.597,Z 290.483,A -85,B 0,C 180,E1 -15095.303,E2 -15095.303} C_VEL
LIN {X 0,Y 319.588,Z 290.487,A -85,B 0,C 180,E1 -15098.047,E2 -15098.047} C_VEL
LIN {X 0,Y 319.681,Z 290.473,A -85,B 0,C 180,E1 -15100.962,E2 -15100.962} C_VEL
LIN {X 0,Y 319.722,Z 290.468,A -85,B 0,C 180,E1 -15105.276,E2 -15105.276} C_VEL
LIN {X 0,Y 319.743,Z 290.465,A -85,B 0,C 180,E1 -15109.872,E2 -15109.872} C_VEL
LIN {X 0,Y 319.903,Z 290.447,A -85,B 0,C 180,E1 -15112.425,E2 -15112.425} C_VEL
LIN {X 0,Y 319.735,Z 290.471,A -85,B 0,C 180,E1 -15114.956,E2 -15114.956} C_VEL
LIN {X 0,Y 319.98,Z 290.437,A -85,B 0,C 180,E1 -15117.482,E2 -15117.482} C_VEL
LIN {X 0,Y 320.139,Z 290.416,A -85,B 0,C 180,E1 -15120,E2 -15120} C_VEL
LIN {X 0,Y 319.979,Z 290.436,A -85,B 0,C 180,E1 -15122.518,E2 -15122.518} C_VEL
LIN {X 0,Y 319.933,Z 290.441,A -85,B 0,C 180,E1 -15126.306,E2 -15126.306} C_VEL
LIN {X 0,Y 319.829,Z 290.455,A -85,B 0,C 180,E1 -15128.848,E2 -15128.848} C_VEL
LIN {X 0,Y 319.675,Z 290.473,A -85,B 0,C 180,E1 -15132.7,E2 -15132.7} C_VEL
LIN {X 0,Y 319.69,Z 290.474,A -85,B 0,C 180,E1 -15135.296,E2 -15135.296} C_VEL
LIN {X 0,Y 319.643,Z 290.479,A -85,B 0,C 180,E1 -15139.257,E2 -15139.257} C_VEL
LIN {X 0,Y 319.553,Z 290.489,A -85,B 0,C 180,E1 -15143.321,E2 -15143.321} C_VEL
LIN {X 0,Y 319.626,Z 290.486,A -85,B 0,C 180,E1 -15146.089,E2 -15146.089} C_VEL
LIN {X 0,Y 319.571,Z 290.487,A -85,B 0,C 180,E1 -15148.935,E2 -15148.935} C_VEL
LIN {X 0,Y 319.522,Z 290.495,A -85,B 0,C 180,E1 -15151.863,E2 -15151.863} C_VEL
LIN {X 0,Y 319.572,Z 290.487,A -85,B 0,C 180,E1 -15155.543,E2 -15155.543} C_VEL
LIN {X 0,Y 319.55,Z 290.491,A -85,B 0,C 180,E1 -15158.011,E2 -15158.011} C_VEL
LIN {X 0,Y 319.519,Z 290.492,A -85,B 0,C 180,E1 -15161.598,E2 -15161.598} C_VEL
LIN {X 0,Y 319.51,Z 290.5,A -85,B 0,C 180,E1 -15164.739,E2 -15164.739} C_VEL
LIN {X 0,Y 319.52,Z 290.495,A -85,B 0,C 180,E1 -15168.404,E2 -15168.404} C_VEL
LIN {X 0,Y 319.538,Z 290.491,A -85,B 0,C 180,E1 -15171.988,E2 -15171.988} C_VEL
LIN {X 0,Y 319.557,Z 290.494,A -85,B 0,C 180,E1 -15175.124,E2 -15175.124} C_VEL
LIN {X 0,Y 319.521,Z 290.493,A -85,B 0,C 180,E1 -15178.138,E2 -15178.138} C_VEL
LIN {X 0,Y 319.569,Z 290.491,A -85,B 0,C 180,E1 -15181.604,E2 -15181.604} C_VEL
LIN {X 0,Y 319.634,Z 290.641,A -85,B 0,C 180,E1 -15182.59,E2 -15182.59} C_VEL
LIN {X 0,Y 321.596,Z 301.12,A -85,B 0,C 180,E1 -15186.068,E2 -15186.068} C_VEL
LIN {X 0,Y 321.763,Z 304.666,A -85,B 0,C 180,E1 -15187.189,E2 -15187.189} C_VEL
LIN {X 0,Y 320.476,Z 316.868,A -85,B 0,C 180,E1 -15190.899,E2 -15190.899} C_VEL
LIN {X 0,Y 324.79,Z 348.918,A -85,B 0,C 180,E1 -15191.89,E2 -15191.89} C_VEL
LIN {X 0,Y 324.075,Z 394.61,A -85,B 0,C 180,E1 -15192.971,E2 -15192.971} C_VEL
LIN {X 0,Y 323.51,Z 404.871,A -85,B 0,C 180,E1 -15193.389,E2 -15193.389} C_VEL
LIN {X 0,Y 322.878,Z 415.551,A -85,B 0,C 180,E1 -15194.05,E2 -15194.05} C_VEL
LIN {X 0,Y 322.045,Z 426.149,A -85,B 0,C 180,E1 -15194.981,E2 -15194.981} C_VEL
LIN {X 0,Y 321.294,Z 434.47,A -85,B 0,C 180,E1 -15195.916,E2 -15195.916} C_VEL
LIN {X 0,Y 320.553,Z 442.354,A -85,B 0,C 180,E1 -15197.014,E2 -15197.014} C_VEL
LIN {X 0,Y 319.808,Z 449.727,A -85,B 0,C 180,E1 -15198.272,E2 -15198.272} C_VEL
LIN {X 0,Y 318.994,Z 457.194,A -85,B 0,C 180,E1 -15199.849,E2 -15199.849} C_VEL
LIN {X 0,Y 318.48,Z 463.031,A -85,B 0,C 180,E1 -15201.434,E2 -15201.434} C_VEL
LIN {X 0,Y 318.102,Z 467.632,A -85,B 0,C 180,E1 -15203.021,E2 -15203.021} C_VEL
LIN {X 0,Y 317.913,Z 470.334,A -85,B 0,C 180,E1 -15204.153,E2 -15204.153} C_VEL
LIN {X 0,Y 317.839,Z 473.832,A -85,B 0,C 180,E1 -15206.197,E2 -15206.197} C_VEL
LIN {X 0,Y 317.765,Z 475.361,A -85,B 0,C 180,E1 -15207.465,E2 -15207.465} C_VEL
LIN {X 0,Y 317.734,Z 476.319,A -85,B 0,C 180,E1 -15208.733,E2 -15208.733} C_VEL
LIN {X 0,Y 317.779,Z 476.712,A -85,B 0,C 180,E1 -15210,E2 -15210} C_VEL
LIN {X 0,Y 317.732,Z 476.632,A -85,B 0,C 180,E1 -15211.267,E2 -15211.267} C_VEL
LIN {X 0,Y 317.764,Z 476.087,A -85,B 0,C 180,E1 -15212.535,E2 -15212.535} C_VEL
LIN {X 0,Y 317.837,Z 475.052,A -85,B 0,C 180,E1 -15213.803,E2 -15213.803} C_VEL
LIN {X 0,Y 317.916,Z 472.125,A -85,B 0,C 180,E1 -15215.852,E2 -15215.852} C_VEL
LIN {X 0,Y 318.321,Z 468.463,A -85,B 0,C 180,E1 -15217.612,E2 -15217.612} C_VEL
LIN {X 0,Y 318.661,Z 465.085,A -85,B 0,C 180,E1 -15218.881,E2 -15218.881} C_VEL
LIN {X 0,Y 319.269,Z 459.816,A -85,B 0,C 180,E1 -15220.463,E2 -15220.463} C_VEL
LIN {X 0,Y 319.956,Z 454.662,A -85,B 0,C 180,E1 -15221.723,E2 -15221.723} C_VEL
LIN {X 0,Y 320.812,Z 448.467,A -85,B 0,C 180,E1 -15222.976,E2 -15222.976} C_VEL
LIN {X 0,Y 321.595,Z 441.969,A -85,B 0,C 180,E1 -15224.07,E2 -15224.07} C_VEL
LIN {X 0,Y 322.562,Z 434.111,A -85,B 0,C 180,E1 -15225.156,E2 -15225.156} C_VEL
LIN {X 0,Y 323.526,Z 425.834,A -85,B 0,C 180,E1 -15226.079,E2 -15226.079} C_VEL
LIN {X 0,Y 324.449,Z 415.336,A -85,B 0,C 180,E1 -15227.003,E2 -15227.003} C_VEL
LIN {X 0,Y 325.346,Z 403.838,A -85,B 0,C 180,E1 -15227.699,E2 -15227.699} C_VEL
LIN {X 0,Y 325.926,Z 393.806,A -85,B 0,C 180,E1 -15228.099,E2 -15228.099} C_VEL
LIN {X 0,Y 326.694,Z 348.706,A -85,B 0,C 180,E1 -15229.18,E2 -15229.18} C_VEL
LIN {X 0,Y 323.06,Z 324.95,A -85,B 0,C 180,E1 -15230.025,E2 -15230.025} C_VEL
LIN {X 0,Y 321.304,Z 315.896,A -85,B 0,C 180,E1 -15230.389,E2 -15230.389} C_VEL
LIN {X 0,Y 322.262,Z 306.722,A -85,B 0,C 180,E1 -15233.112,E2 -15233.112} C_VEL
LIN {X 0,Y 322.228,Z 303.88,A -85,B 0,C 180,E1 -15233.99,E2 -15233.99} C_VEL
LIN {X 0,Y 320.198,Z 293.465,A -85,B 0,C 180,E1 -15237.446,E2 -15237.446} C_VEL
LIN {X 0,Y 319.571,Z 290.492,A -85,B 0,C 180,E1 -15238.523,E2 -15238.523} C_VEL
LIN {X 0,Y 319.52,Z 290.494,A -85,B 0,C 180,E1 -15241.862,E2 -15241.862} C_VEL
LIN {X 0,Y 319.576,Z 290.492,A -85,B 0,C 180,E1 -15245.542,E2 -15245.542} C_VEL
LIN {X 0,Y 319.552,Z 290.497,A -85,B 0,C 180,E1 -15248.009,E2 -15248.009} C_VEL
LIN {X 0,Y 319.52,Z 290.499,A -85,B 0,C 180,E1 -15251.596,E2 -15251.596} C_VEL
LIN {X 0,Y 319.482,Z 290.502,A -85,B 0,C 180,E1 -15255.256,E2 -15255.256} C_VEL
LIN {X 0,Y 319.521,Z 290.492,A -85,B 0,C 180,E1 -15258.711,E2 -15258.711} C_VEL
LIN {X 0,Y 319.554,Z 290.485,A -85,B 0,C 180,E1 -15262.347,E2 -15262.347} C_VEL
LIN {X 0,Y 319.552,Z 290.492,A -85,B 0,C 180,E1 -15265.123,E2 -15265.123} C_VEL
LIN {X 0,Y 319.562,Z 290.487,A -85,B 0,C 180,E1 -15269.057,E2 -15269.057} C_VEL
LIN {X 0,Y 319.599,Z 290.474,A -85,B 0,C 180,E1 -15272.497,E2 -15272.497} C_VEL
LIN {X 0,Y 319.594,Z 290.485,A -85,B 0,C 180,E1 -15275.303,E2 -15275.303} C_VEL
LIN {X 0,Y 319.592,Z 290.478,A -85,B 0,C 180,E1 -15279.4,E2 -15279.4} C_VEL
LIN {X 0,Y 319.648,Z 290.482,A -85,B 0,C 180,E1 -15282.073,E2 -15282.073} C_VEL
LIN {X 0,Y 319.722,Z 290.464,A -85,B 0,C 180,E1 -15286.008,E2 -15286.008} C_VEL
LIN {X 0,Y 319.742,Z 290.459,A -85,B 0,C 180,E1 -15289.873,E2 -15289.873} C_VEL
LIN {X 0,Y 319.903,Z 290.442,A -85,B 0,C 180,E1 -15292.426,E2 -15292.426} C_VEL
LIN {X 0,Y 319.733,Z 290.463,A -85,B 0,C 180,E1 -15294.956,E2 -15294.956} C_VEL
LIN {X 0,Y 319.978,Z 290.43,A -85,B 0,C 180,E1 -15297.482,E2 -15297.482} C_VEL
LIN {X 0,Y 320.139,Z 290.415,A -85,B 0,C 180,E1 -15300,E2 -15300} C_VEL
LIN {X 0,Y 319.978,Z 290.426,A -85,B 0,C 180,E1 -15302.518,E2 -15302.518} C_VEL
LIN {X 0,Y 319.883,Z 290.445,A -85,B 0,C 180,E1 -15306.465,E2 -15306.465} C_VEL
LIN {X 0,Y 319.742,Z 290.467,A -85,B 0,C 180,E1 -15310.128,E2 -15310.128} C_VEL
LIN {X 0,Y 319.722,Z 290.471,A -85,B 0,C 180,E1 -15314.724,E2 -15314.724} C_VEL
LIN {X 0,Y 319.681,Z 290.479,A -85,B 0,C 180,E1 -15319.038,E2 -15319.038} C_VEL
LIN {X 0,Y 319.562,Z 290.493,A -85,B 0,C 180,E1 -15323.32,E2 -15323.32} C_VEL
LIN {X 0,Y 319.627,Z 290.483,A -85,B 0,C 180,E1 -15326.089,E2 -15326.089} C_VEL
LIN {X 0,Y 319.582,Z 290.485,A -85,B 0,C 180,E1 -15328.935,E2 -15328.935} C_VEL
LIN {X 0,Y 319.525,Z 290.498,A -85,B 0,C 180,E1 -15331.863,E2 -15331.863} C_VEL
LIN {X 0,Y 319.573,Z 290.486,A -85,B 0,C 180,E1 -15335.544,E2 -15335.544} C_VEL
LIN {X 0,Y 319.643,Z 290.627,A -85,B 0,C 180,E1 -15338.5,E2 -15338.5} C_VEL
LIN {X 0,Y 321.613,Z 300.148,A -85,B 0,C 180,E1 -15341.692,E2 -15341.692} C_VEL
LIN {X 0,Y 323.936,Z 308.33,A -85,B 0,C 180,E1 -15342.072,E2 -15342.072} C_VEL
LIN {X 0,Y 327.289,Z 325.616,A -85,B 0,C 180,E1 -15342.742,E2 -15342.742} C_VEL
LIN {X 0,Y 326.089,Z 377.452,A -85,B 0,C 180,E1 -15343.963,E2 -15343.963} C_VEL
LIN {X 0,Y 325.61,Z 387.831,A -85,B 0,C 180,E1 -15344.393,E2 -15344.393} C_VEL
LIN {X 0,Y 324.89,Z 399.761,A -85,B 0,C 180,E1 -15345.167,E2 -15345.167} C_VEL
LIN {X 0,Y 324.148,Z 408.188,A -85,B 0,C 180,E1 -15345.907,E2 -15345.907} C_VEL
LIN {X 0,Y 323.334,Z 416.216,A -85,B 0,C 180,E1 -15346.791,E2 -15346.791} C_VEL
LIN {X 0,Y 322.31,Z 424.612,A -85,B 0,C 180,E1 -15347.939,E2 -15347.939} C_VEL
LIN {X 0,Y 321.489,Z 431.071,A -85,B 0,C 180,E1 -15349.02,E2 -15349.02} C_VEL
LIN {X 0,Y 320.772,Z 436.37,A -85,B 0,C 180,E1 -15350.071,E2 -15350.071} C_VEL
LIN {X 0,Y 320.111,Z 441.445,A -85,B 0,C 180,E1 -15351.267,E2 -15351.267} C_VEL
LIN {X 0,Y 319.317,Z 447.123,A -85,B 0,C 180,E1 -15352.927,E2 -15352.927} C_VEL
LIN {X 0,Y 318.675,Z 451.781,A -85,B 0,C 180,E1 -15354.686,E2 -15354.686} C_VEL
LIN {X 0,Y 318.289,Z 455.314,A -85,B 0,C 180,E1 -15356.496,E2 -15356.496} C_VEL
LIN {X 0,Y 317.964,Z 457.288,A -85,B 0,C 180,E1 -15357.964,E2 -15357.964} C_VEL
LIN {X 0,Y 317.703,Z 458.702,A -85,B 0,C 180,E1 -15359.625,E2 -15359.625} C_VEL
LIN {X 0,Y 317.575,Z 459.143,A -85,B 0,C 180,E1 -15360.866,E2 -15360.866} C_VEL
LIN {X 0,Y 317.541,Z 459.096,A -85,B 0,C 180,E1 -15362.305,E2 -15362.305} C_VEL
LIN {X 0,Y 317.585,Z 458.423,A -85,B 0,C 180,E1 -15363.732,E2 -15363.732} C_VEL
LIN {X 0,Y 317.745,Z 457.122,A -85,B 0,C 180,E1 -15365.151,E2 -15365.151} C_VEL
LIN {X 0,Y 317.969,Z 455.187,A -85,B 0,C 180,E1 -15366.557,E2 -15366.557} C_VEL
LIN {X 0,Y 318.258,Z 452.36,A -85,B 0,C 180,E1 -15368.045,E2 -15368.045} C_VEL
LIN {X 0,Y 318.657,Z 448.234,A -85,B 0,C 180,E1 -15369.674,E2 -15369.674} C_VEL
LIN {X 0,Y 319.144,Z 443.13,A -85,B 0,C 180,E1 -15371.249,E2 -15371.249} C_VEL
LIN {X 0,Y 319.612,Z 438.61,A -85,B 0,C 180,E1 -15372.402,E2 -15372.402} C_VEL
LIN {X 0,Y 320.285,Z 432.189,A -85,B 0,C 180,E1 -15373.746,E2 -15373.746} C_VEL
LIN {X 0,Y 320.963,Z 425.323,A -85,B 0,C 180,E1 -15374.929,E2 -15374.929} C_VEL
LIN {X 0,Y 321.672,Z 418.273,A -85,B 0,C 180,E1 -15375.933,E2 -15375.933} C_VEL
LIN {X 0,Y 322.457,Z 409.641,A -85,B 0,C 180,E1 -15376.931,E2 -15376.931} C_VEL
LIN {X 0,Y 323.146,Z 400.01,A -85,B 0,C 180,E1 -15377.809,E2 -15377.809} C_VEL
LIN {X 0,Y 323.74,Z 389.319,A -85,B 0,C 180,E1 -15378.537,E2 -15378.537} C_VEL
LIN {X 0,Y 324.188,Z 378.246,A -85,B 0,C 180,E1 -15379.026,E2 -15379.026} C_VEL
LIN {X 0,Y 324.637,Z 354.256,A -85,B 0,C 180,E1 -15379.618,E2 -15379.618} C_VEL
LIN {X 0,Y 325.075,Z 324.044,A -85,B 0,C 180,E1 -15380.309,E2 -15380.309} C_VEL
LIN {X 0,Y 320.847,Z 300.082,A -85,B 0,C 180,E1 -15381.125,E2 -15381.125} C_VEL
LIN {X 0,Y 320.756,Z 296.238,A -85,B 0,C 180,E1 -15382.446,E2 -15382.446} C_VEL
LIN {X 0,Y 319.821,Z 290.461,A -85,B 0,C 180,E1 -15384.562,E2 -15384.562} C_VEL
LIN {X 0,Y 319.991,Z 290.438,A -85,B 0,C 180,E1 -15387.483,E2 -15387.483} C_VEL
LIN {X 0,Y 320.151,Z 290.42,A -85,B 0,C 180,E1 -15390,E2 -15390} C_VEL
LIN {X 0,Y 319.991,Z 290.436,A -85,B 0,C 180,E1 -15392.518,E2 -15392.518} C_VEL
LIN {X 0,Y 319.913,Z 290.448,A -85,B 0,C 180,E1 -15396.306,E2 -15396.306} C_VEL
LIN {X 0,Y 319.753,Z 290.469,A -85,B 0,C 180,E1 -15400.127,E2 -15400.127} C_VEL
LIN {X 0,Y 319.733,Z 290.468,A -85,B 0,C 180,E1 -15403.992,E2 -15403.992} C_VEL
LIN {X 0,Y 319.625,Z 290.481,A -85,B 0,C 180,E1 -15407.928,E2 -15407.928} C_VEL
LIN {X 0,Y 319.568,Z 290.486,A -85,B 0,C 180,E1 -15411.954,E2 -15411.954} C_VEL
LIN {X 0,Y 319.618,Z 290.481,A -85,B 0,C 180,E1 -15416.089,E2 -15416.089} C_VEL
LIN {X 0,Y 319.589,Z 290.491,A -85,B 0,C 180,E1 -15418.933,E2 -15418.933} C_VEL
LIN {X 0,Y 319.531,Z 290.492,A -85,B 0,C 180,E1 -15421.861,E2 -15421.861} C_VEL
LIN {X 0,Y 319.577,Z 290.488,A -85,B 0,C 180,E1 -15425.542,E2 -15425.542} C_VEL
LIN {X 0,Y 319.555,Z 290.491,A -85,B 0,C 180,E1 -15429.668,E2 -15429.668} C_VEL
LIN {X 0,Y 319.56,Z 290.494,A -85,B 0,C 180,E1 -15433.468,E2 -15433.468} C_VEL
LIN {X 0,Y 319.6,Z 290.484,A -85,B 0,C 180,E1 -15437.024,E2 -15437.024} C_VEL
LIN {X 0,Y 319.576,Z 290.486,A -85,B 0,C 180,E1 -15440.406,E2 -15440.406} C_VEL
LIN {X 0,Y 318.856,Z 290.579,A -85,B 0,C 180,E1 -15441.458,E2 -15441.458} C_VEL
LIN {X 0,Y 315.98,Z 290.934,A -85,B 0,C 180,E1 -15443.171,E2 -15443.171} C_VEL
LIN {X 0,Y 313.584,Z 291.236,A -85,B 0,C 180,E1 -15444.56,E2 -15444.56} C_VEL
LIN {X 0,Y 312.576,Z 291.361,A -85,B 0,C 180,E1 -15445.635,E2 -15445.635} C_VEL
LIN {X 0,Y 312.502,Z 291.369,A -85,B 0,C 180,E1 -15445.999,E2 -15445.999} C_VEL
LIN {X 0,Y 312.538,Z 291.366,A -85,B 0,C 180,E1 -15450.349,E2 -15450.349} C_VEL
LIN {X 0,Y 312.596,Z 291.36,A -85,B 0,C 180,E1 -15454.064,E2 -15454.064} C_VEL
LIN {X 0,Y 312.58,Z 291.356,A -85,B 0,C 180,E1 -15457.528,E2 -15457.528} C_VEL
LIN {X 0,Y 312.63,Z 291.35,A -85,B 0,C 180,E1 -15461.656,E2 -15461.656} C_VEL
LIN {X 0,Y 312.685,Z 291.344,A -85,B 0,C 180,E1 -15465.686,E2 -15465.686} C_VEL
LIN {X 0,Y 312.689,Z 291.344,A -85,B 0,C 180,E1 -15469.641,E2 -15469.641} C_VEL
LIN {X 0,Y 312.844,Z 291.325,A -85,B 0,C 180,E1 -15472.253,E2 -15472.253} C_VEL
LIN {X 0,Y 312.705,Z 291.345,A -85,B 0,C 180,E1 -15474.842,E2 -15474.842} C_VEL
LIN {X 0,Y 312.98,Z 291.309,A -85,B 0,C 180,E1 -15478.713,E2 -15478.713} C_VEL
LIN {X 0,Y 312.982,Z 291.312,A -85,B 0,C 180,E1 -15481.287,E2 -15481.287} C_VEL
LIN {X 0,Y 312.705,Z 291.347,A -85,B 0,C 180,E1 -15485.158,E2 -15485.158} C_VEL
LIN {X 0,Y 312.843,Z 291.326,A -85,B 0,C 180,E1 -15487.746,E2 -15487.746} C_VEL
LIN {X 0,Y 312.662,Z 291.351,A -85,B 0,C 180,E1 -15491.671,E2 -15491.671} C_VEL
LIN {X 0,Y 312.691,Z 291.344,A -85,B 0,C 180,E1 -15494.888,E2 -15494.888} C_VEL
LIN {X 0,Y 312.6,Z 291.356,A -85,B 0,C 180,E1 -15499.225,E2 -15499.225} C_VEL
LIN {X 0,Y 312.519,Z 291.365,A -85,B 0,C 180,E1 -15502.781,E2 -15502.781} C_VEL
LIN {X 0,Y 312.594,Z 291.361,A -85,B 0,C 180,E1 -15505.936,E2 -15505.936} C_VEL
LIN {X 0,Y 312.53,Z 291.365,A -85,B 0,C 180,E1 -15509.651,E2 -15509.651} C_VEL
LIN {X 0,Y 312.512,Z 291.367,A -85,B 0,C 180,E1 -15513.689,E2 -15513.689} C_VEL
LIN {X 0,Y 312.518,Z 291.365,A -85,B 0,C 180,E1 -15517.386,E2 -15517.386} C_VEL
LIN {X 0,Y 312.484,Z 291.372,A -85,B 0,C 180,E1 -15520.71,E2 -15520.71} C_VEL
LIN {X 0,Y 312.467,Z 291.373,A -85,B 0,C 180,E1 -15524.207,E2 -15524.207} C_VEL
LIN {X 0,Y 312.48,Z 291.37,A -85,B 0,C 180,E1 -15527.919,E2 -15527.919} C_VEL
LIN {X 0,Y 312.493,Z 291.374,A -85,B 0,C 180,E1 -15530.972,E2 -15530.972} C_VEL
LIN {X 0,Y 312.528,Z 291.364,A -85,B 0,C 180,E1 -15534.221,E2 -15534.221} C_VEL
LIN {X 0,Y 312.498,Z 291.372,A -85,B 0,C 180,E1 -15537.334,E2 -15537.334} C_VEL
LIN {X 0,Y 312.504,Z 291.373,A -85,B 0,C 180,E1 -15541.292,E2 -15541.292} C_VEL
LIN {X 0,Y 312.558,Z 291.464,A -85,B 0,C 180,E1 -15542.325,E2 -15542.325} C_VEL
LIN {X 0,Y 314.564,Z 302.098,A -85,B 0,C 180,E1 -15545.938,E2 -15545.938} C_VEL
LIN {X 0,Y 314.768,Z 305.37,A -85,B 0,C 180,E1 -15547.001,E2 -15547.001} C_VEL
LIN {X 0,Y 313.575,Z 316.748,A -85,B 0,C 180,E1 -15550.526,E2 -15550.526} C_VEL
LIN {X 0,Y 318.011,Z 350.224,A -85,B 0,C 180,E1 -15551.582,E2 -15551.582} C_VEL
LIN {X 0,Y 317.222,Z 394.449,A -85,B 0,C 180,E1 -15552.65,E2 -15552.65} C_VEL
